C03641=1096.740,305.564,-82.247,178.244,19.160,152.472
C03642=1096.746,305.813,-82.279,178.248,19.162,152.472
C03643=1096.752,306.060,-82.310,178.251,19.165,152.472
C03644=1096.757,306.309,-82.341,178.254,19.167,152.472
C03645=1096.763,306.556,-82.371,178.257,19.170,152.472
C03646=1096.769,306.805,-82.402,178.261,19.172,152.472
C03647=1096.775,307.052,-82.434,178.264,19.175,152.472
C03648=1096.780,307.301,-82.464,178.267,19.177,152.472
C03649=1096.786,307.548,-82.495,178.270,19.180,152.472
C03650=1096.792,307.797,-82.527,178.274,19.183,152.472
C03651=1096.797,308.044,-82.557,178.277,19.185,152.472
C03652=1096.802,308.293,-82.588,178.280,19.188,152.472
C03653=1096.808,308.540,-82.620,178.283,19.190,152.472
C03654=1096.814,308.789,-82.651,178.286,19.193,152.472
C03655=1096.819,309.037,-82.681,178.290,19.195,152.472
C03656=1096.825,309.284,-82.713,178.293,19.197,152.472
C03657=1096.831,309.533,-82.744,178.296,19.200,152.472
C03658=1096.837,309.780,-82.775,178.300,19.203,152.472
C03659=1096.842,310.028,-82.806,178.303,19.206,152.472
C03660=1096.848,310.276,-82.838,178.306,19.208,152.472
C03661=1096.854,310.524,-82.868,178.309,19.211,152.472
C03662=1096.860,310.772,-82.900,178.312,19.213,152.472
C03663=1096.866,311.020,-82.931,178.315,19.215,152.472
C03664=1096.871,311.268,-82.962,178.318,19.218,152.472
C03665=1096.877,311.517,-82.994,178.322,19.221,152.473
C03666=1096.883,311.764,-83.025,178.325,19.223,152.472
C03667=1096.888,312.012,-83.056,178.328,19.226,152.473
C03668=1096.894,312.260,-83.088,178.332,19.229,152.473
C03669=1096.900,312.507,-83.119,178.335,19.231,152.473
C03670=1096.906,312.756,-83.150,178.338,19.234,152.473
C03671=1096.912,313.003,-83.181,178.341,19.237,152.473
C03672=1096.918,313.252,-83.213,178.344,19.239,152.473
C03673=1096.923,313.500,-83.244,178.347,19.241,152.473
C03674=1096.929,313.747,-83.276,178.351,19.244,152.473
C03675=1096.935,313.995,-83.307,178.354,19.247,152.473
C03676=1096.940,314.243,-83.338,178.357,19.249,152.473
C03677=1096.946,314.491,-83.370,178.361,19.252,152.473
C03678=1096.953,314.739,-83.401,178.364,19.255,152.473
C03679=1096.959,314.987,-83.433,178.367,19.258,152.473
C03680=1096.964,315.235,-83.464,178.370,19.260,152.473
C03681=1096.970,315.483,-83.496,178.373,19.263,152.473
C03682=1096.975,315.731,-83.528,178.376,19.265,152.473
C03683=1096.983,316.120,-83.577,178.382,19.270,152.473
C03684=1096.993,316.508,-83.626,178.386,19.274,152.473
C03685=1097.002,316.897,-83.677,178.391,19.279,152.474
C03686=1097.010,317.286,-83.726,178.396,19.283,152.474
C03687=1097.016,317.534,-83.758,178.399,19.286,152.474
C03688=1097.022,317.782,-83.790,178.403,19.289,152.474
C03689=1097.027,318.029,-83.822,178.406,19.291,152.474
C03690=1097.033,318.277,-83.854,178.409,19.295,152.474
C03691=1097.038,318.525,-83.886,178.412,19.297,152.474
C03692=1097.044,318.774,-83.918,178.415,19.300,152.474
C03693=1097.049,319.021,-83.950,178.418,19.303,152.474
C03694=1097.055,319.269,-83.982,178.422,19.306,152.474
C03695=1097.061,319.517,-84.013,178.425,19.308,152.475
C03696=1097.067,319.765,-84.045,178.428,19.311,152.475
C03697=1097.072,320.012,-84.077,178.431,19.314,152.475
C03698=1097.078,320.261,-84.109,178.434,19.317,152.475
C03699=1097.083,320.508,-84.141,178.438,19.320,152.475
C03700=1097.089,320.756,-84.173,178.441,19.323,152.475
C03701=1097.094,321.004,-84.205,178.444,19.326,152.475
C03702=1097.100,321.252,-84.237,178.446,19.329,152.475
C03703=1097.105,321.500,-84.269,178.450,19.331,152.475
C03704=1097.111,321.748,-84.301,178.453,19.335,152.476
C03705=1097.117,321.996,-84.332,178.456,19.337,152.476
C03706=1097.123,322.243,-84.365,178.459,19.340,152.476
C03707=1097.128,322.492,-84.398,178.462,19.343,152.476
C03708=1097.134,322.739,-84.429,178.465,19.346,152.476
C03709=1097.140,322.988,-84.461,178.469,19.349,152.476
C03710=1097.145,323.235,-84.493,178.472,19.352,152.476
C03711=1097.151,323.483,-84.526,178.475,19.355,152.476
C03712=1097.156,323.731,-84.558,178.478,19.357,152.477
C03713=1097.162,323.979,-84.590,178.481,19.360,152.477
C03714=1097.168,324.227,-84.622,178.485,19.364,152.477
C03715=1097.174,324.474,-84.655,178.488,19.366,152.477
C03716=1097.180,324.722,-84.687,178.491,19.369,152.477
C03717=1097.185,324.971,-84.719,178.494,19.372,152.477
C03718=1097.191,325.218,-84.752,178.498,19.375,152.477
C03719=1097.196,325.466,-84.784,178.500,19.379,152.478
C03720=1097.202,325.714,-84.816,178.504,19.381,152.478
C03721=1097.208,325.962,-84.849,178.507,19.384,152.478
C03722=1097.214,326.210,-84.881,178.510,19.388,152.478
C03723=1097.220,326.457,-84.913,178.513,19.390,152.478
C03724=1097.225,326.705,-84.946,178.516,19.393,152.478
C03725=1097.231,326.954,-84.978,178.519,19.396,152.478
C03726=1097.237,327.200,-85.010,178.523,19.399,152.478
C03727=1097.243,327.449,-85.042,178.526,19.402,152.479
C03728=1097.248,327.697,-85.076,178.529,19.405,152.479
C03729=1097.254,327.945,-85.108,178.532,19.408,152.479
C03730=1097.260,328.192,-85.140,178.536,19.411,152.479
C03731=1097.265,328.440,-85.173,178.539,19.414,152.479
C03732=1097.271,328.688,-85.206,178.541,19.417,152.479
C03733=1097.278,328.935,-85.238,178.544,19.420,152.479
C03734=1097.283,329.184,-85.271,178.548,19.423,152.480
C03735=1097.292,329.565,-85.320,178.553,19.428,152.480
C03736=1097.301,329.947,-85.371,178.558,19.433,152.480
C03737=1097.310,330.328,-85.422,178.563,19.438,152.480
C03738=1097.319,330.711,-85.472,178.567,19.442,152.481
C03739=1097.325,330.958,-85.504,178.570,19.445,152.481
C03740=1097.330,331.206,-85.537,178.574,19.448,152.481
C03741=1097.336,331.454,-85.570,178.577,19.451,152.481
C03742=1097.342,331.702,-85.603,178.580,19.454,152.481
C03743=1097.348,331.949,-85.636,178.584,19.458,152.481
C03744=1097.354,332.197,-85.668,178.586,19.461,152.482
C03745=1097.360,332.445,-85.701,178.589,19.464,152.482
C03746=1097.365,332.692,-85.734,178.593,19.467,152.482
C03747=1097.371,332.940,-85.767,178.596,19.470,152.482
C03748=1097.376,333.189,-85.800,178.599,19.473,152.482
C03749=1097.382,333.436,-85.833,178.602,19.477,152.483
C03750=1097.388,333.684,-85.866,178.605,19.480,152.483
C03751=1097.394,333.932,-85.899,178.608,19.483,152.483
C03752=1097.400,334.180,-85.932,178.612,19.487,152.483
C03753=1097.405,334.427,-85.965,178.615,19.489,152.483
C03754=1097.410,334.675,-85.998,178.618,19.493,152.484
C03755=1097.417,334.922,-86.031,178.621,19.496,152.484
C03756=1097.422,335.170,-86.064,178.624,19.499,152.484
C03757=1097.428,335.418,-86.097,178.627,19.502,152.484
C03758=1097.433,335.667,-86.130,178.630,19.506,152.485
C03759=1097.439,335.914,-86.163,178.633,19.509,152.485
C03760=1097.445,336.162,-86.196,178.636,19.512,152.485
C03761=1097.450,336.410,-86.229,178.640,19.516,152.485
C03762=1097.456,336.656,-86.263,178.643,19.519,152.485
C03763=1097.462,336.904,-86.296,178.646,19.523,152.486
C03764=1097.467,337.152,-86.329,178.649,19.526,152.486
C03765=1097.473,337.400,-86.363,178.652,19.529,152.486
C03766=1097.479,337.648,-86.395,178.655,19.533,152.486
C03767=1097.485,337.895,-86.429,178.658,19.536,152.487
C03768=1097.490,338.143,-86.462,178.661,19.539,152.487
C03769=1097.496,338.391,-86.495,178.665,19.542,152.487
C03770=1097.502,338.639,-86.528,178.668,19.546,152.487
C03771=1097.508,338.886,-86.562,178.671,19.550,152.488
C03772=1097.514,339.134,-86.595,178.674,19.553,152.488
C03773=1097.519,339.382,-86.629,178.677,19.556,152.488
C03774=1097.525,339.630,-86.662,178.680,19.560,152.488
C03775=1097.530,339.878,-86.695,178.683,19.563,152.489
C03776=1097.536,340.125,-86.730,178.686,19.567,152.489
C03777=1097.542,340.373,-86.763,178.689,19.570,152.489
C03778=1097.547,340.621,-86.796,178.693,19.573,152.489
C03779=1097.553,340.869,-86.830,178.696,19.577,152.490
C03780=1097.559,341.116,-86.863,178.698,19.580,152.490
C03781=1097.565,341.364,-86.896,178.702,19.584,152.490
C03782=1097.571,341.612,-86.930,178.705,19.587,152.491
C03783=1097.576,341.859,-86.964,178.708,19.591,152.491
C03784=1097.582,342.107,-86.997,178.711,19.594,152.491
C03785=1097.588,342.354,-87.031,178.714,19.598,152.492
C03786=1097.593,342.602,-87.064,178.717,19.601,152.492
C03787=1097.602,342.979,-87.116,178.722,19.607,152.492
C03788=1097.611,343.353,-87.167,178.727,19.612,152.493
C03789=1097.619,343.729,-87.218,178.731,19.617,152.493
C03790=1097.629,344.105,-87.269,178.736,19.623,152.494
C03791=1097.634,344.353,-87.304,178.740,19.626,152.494
C03792=1097.640,344.601,-87.337,178.742,19.630,152.494
C03793=1097.645,344.848,-87.371,178.746,19.634,152.494
C03794=1097.651,345.096,-87.404,178.748,19.637,152.495
C03795=1097.657,345.343,-87.438,178.751,19.641,152.495
C03796=1097.662,345.591,-87.472,178.755,19.644,152.495
C03797=1097.668,345.838,-87.506,178.757,19.648,152.496
C03798=1097.674,346.085,-87.540,178.761,19.652,152.496
C03799=1097.680,346.334,-87.573,178.764,19.655,152.496
C03800=1097.685,346.582,-87.608,178.767,19.659,152.497
C03801=1097.691,346.829,-87.642,178.770,19.663,152.497
C03802=1097.697,347.077,-87.675,178.773,19.666,152.497
C03803=1097.703,347.324,-87.710,178.776,19.670,152.498
C03804=1097.708,347.571,-87.744,178.779,19.674,152.498
C03805=1097.714,347.819,-87.778,178.782,19.677,152.499
C03806=1097.720,348.068,-87.812,178.785,19.681,152.499
C03807=1097.726,348.315,-87.846,178.789,19.685,152.499
C03808=1097.731,348.562,-87.880,178.791,19.689,152.500
C03809=1097.737,348.809,-87.914,178.795,19.693,152.500
C03810=1097.742,349.058,-87.948,178.798,19.696,152.500
C03811=1097.748,349.305,-87.982,178.801,19.700,152.501
C03812=1097.754,349.553,-88.017,178.804,19.704,152.501
C03813=1097.760,349.801,-88.051,178.807,19.708,152.501
C03814=1097.765,350.048,-88.085,178.810,19.712,152.502
C03815=1097.771,350.295,-88.119,178.813,19.716,152.502
C03816=1097.776,350.543,-88.154,178.816,19.719,152.503
C03817=1097.783,350.791,-88.188,178.819,19.723,152.503
C03818=1097.789,351.038,-88.222,178.822,19.727,152.503
C03819=1097.794,351.286,-88.257,178.825,19.731,152.504
C03820=1097.800,351.533,-88.291,178.828,19.735,152.504
C03821=1097.806,351.781,-88.326,178.831,19.738,152.504
C03822=1097.811,352.028,-88.360,178.834,19.742,152.505
C03823=1097.817,352.276,-88.394,178.837,19.746,152.505
C03824=1097.823,352.523,-88.428,178.840,19.750,152.506
C03825=1097.829,352.771,-88.463,178.843,19.754,152.506
C03826=1097.835,353.019,-88.497,178.846,19.758,152.506
C03827=1097.841,353.266,-88.531,178.850,19.762,152.507
C03828=1097.846,353.513,-88.566,178.852,19.766,152.507
C03829=1097.852,353.761,-88.600,178.856,19.770,152.508
C03830=1097.857,354.009,-88.635,178.858,19.773,152.508
C03831=1097.863,354.256,-88.669,178.862,19.777,152.508
C03832=1097.869,354.504,-88.705,178.865,19.782,152.509
C03833=1097.875,354.751,-88.739,178.867,19.785,152.509
C03834=1097.880,354.999,-88.774,178.871,19.789,152.510
C03835=1097.886,355.246,-88.808,178.873,19.793,152.510
C03836=1097.892,355.494,-88.843,178.877,19.798,152.511
C03837=1097.897,355.741,-88.878,178.880,19.802,152.511
C03838=1097.903,355.989,-88.912,178.883,19.806,152.512
C03839=1097.911,356.367,-88.965,178.887,19.812,152.512
C03840=1097.921,356.745,-89.018,178.891,19.818,152.513
C03841=1097.930,357.123,-89.071,178.897,19.825,152.514
C03842=1097.938,357.501,-89.125,178.902,19.831,152.514
C03843=1097.944,357.749,-89.160,178.904,19.835,152.515
C03844=1097.950,357.996,-89.194,178.907,19.839,152.515
C03845=1097.955,358.244,-89.229,178.911,19.843,152.516
C03846=1097.962,358.491,-89.264,178.913,19.847,152.516
C03847=1097.967,358.738,-89.299,178.916,19.851,152.517
C03848=1097.973,358.986,-89.334,178.920,19.856,152.517
C03849=1097.979,359.233,-89.369,178.922,19.860,152.518
C03850=1097.985,359.481,-89.404,178.925,19.864,152.518
C03851=1097.990,359.728,-89.439,178.929,19.868,152.519
C03852=1097.997,359.976,-89.474,178.931,19.872,152.519
C03853=1098.002,360.223,-89.509,178.934,19.877,152.520
C03854=1098.007,360.470,-89.544,178.938,19.881,152.520
C03855=1098.013,360.719,-89.579,178.940,19.885,152.521
C03856=1098.019,360.965,-89.614,178.943,19.889,152.521
C03857=1098.025,361.213,-89.650,178.946,19.894,152.522
C03858=1098.030,361.461,-89.684,178.949,19.898,152.522
C03859=1098.036,361.708,-89.720,178.952,19.902,152.523
C03860=1098.042,361.955,-89.755,178.955,19.907,152.523
C03861=1098.048,362.203,-89.789,178.958,19.911,152.524
C03862=1098.054,362.450,-89.825,178.961,19.915,152.524
C03863=1098.059,362.697,-89.860,178.964,19.920,152.525
C03864=1098.065,362.945,-89.895,178.967,19.924,152.525
C03865=1098.070,363.192,-89.931,178.969,19.928,152.526
C03866=1098.077,363.440,-89.966,178.973,19.932,152.526
C03867=1098.082,363.687,-90.001,178.976,19.937,152.527
C03868=1098.088,363.934,-90.037,178.979,19.941,152.527
C03869=1098.093,364.182,-90.072,178.982,19.945,152.528
C03870=1098.100,364.430,-90.107,178.984,19.950,152.529
C03871=1098.105,364.677,-90.143,178.988,19.955,152.529
C03872=1098.111,364.924,-90.179,178.991,19.959,152.530
C03873=1098.117,365.171,-90.213,178.993,19.963,152.530
C03874=1098.123,365.419,-90.249,178.996,19.968,152.531
C03875=1098.129,365.666,-90.284,178.999,19.973,152.531
C03876=1098.135,365.913,-90.320,179.003,19.977,152.532
C03877=1098.141,366.161,-90.356,179.005,19.981,152.532
C03878=1098.146,366.409,-90.391,179.008,19.986,152.533
C03879=1098.152,366.656,-90.426,179.011,19.990,152.534
C03880=1098.158,366.903,-90.462,179.014,19.995,152.534
C03881=1098.163,367.151,-90.499,179.017,19.999,152.535
C03882=1098.168,367.398,-90.534,179.020,20.004,152.535
C03883=1098.174,367.645,-90.570,179.023,20.009,152.536
C03884=1098.180,367.892,-90.605,179.026,20.014,152.537
C03885=1098.186,368.140,-90.641,179.029,20.019,152.537
C03886=1098.191,368.387,-90.676,179.031,20.022,152.538
C03887=1098.197,368.635,-90.712,179.034,20.027,152.539
C03888=1098.203,368.882,-90.747,179.037,20.032,152.539
C03889=1098.209,369.129,-90.783,179.040,20.037,152.540
C03890=1098.215,369.377,-90.819,179.043,20.042,152.540
C03891=1098.223,369.770,-90.876,179.047,20.049,152.541
C03892=1098.232,370.163,-90.933,179.052,20.056,152.542
C03893=1098.242,370.556,-90.990,179.057,20.064,152.543
C03894=1098.251,370.949,-91.047,179.061,20.072,152.545
C03895=1098.256,371.197,-91.083,179.064,20.076,152.545
C03896=1098.263,371.444,-91.119,179.067,20.081,152.546
C03897=1098.268,371.691,-91.155,179.070,20.086,152.546
C03898=1098.274,371.938,-91.191,179.073,20.091,152.547
C03899=1098.280,372.185,-91.227,179.076,20.096,152.548
C03900=1098.285,372.433,-91.263,179.078,20.100,152.548
C03901=1098.291,372.680,-91.299,179.081,20.105,152.549
C03902=1098.297,372.927,-91.335,179.084,20.110,152.550
C03903=1098.304,373.174,-91.372,179.087,20.115,152.550
C03904=1098.309,373.421,-91.407,179.090,20.120,152.551
C03905=1098.315,373.669,-91.443,179.093,20.125,152.552
C03906=1098.321,373.916,-91.480,179.096,20.130,152.553
C03907=1098.326,374.163,-91.515,179.099,20.135,152.553
C03908=1098.333,374.410,-91.552,179.101,20.139,152.554
C03909=1098.338,374.658,-91.589,179.104,20.144,152.555
C03910=1098.344,374.906,-91.624,179.107,20.149,152.555
C03911=1098.349,375.152,-91.661,179.110,20.154,152.556
C03912=1098.355,375.400,-91.697,179.113,20.159,152.557
C03913=1098.362,375.647,-91.733,179.116,20.164,152.558
C03914=1098.366,375.894,-91.769,179.119,20.169,152.558
C03915=1098.373,376.141,-91.806,179.122,20.175,152.559
C03916=1098.378,376.389,-91.843,179.125,20.180,152.560
C03917=1098.384,376.636,-91.878,179.127,20.185,152.561
C03918=1098.389,376.883,-91.915,179.130,20.190,152.561
C03919=1098.396,377.130,-91.951,179.133,20.195,152.562
C03920=1098.401,377.377,-91.988,179.135,20.200,152.563
C03921=1098.407,377.625,-92.024,179.138,20.205,152.564
C03922=1098.412,377.872,-92.061,179.141,20.210,152.564
C03923=1098.419,378.119,-92.097,179.144,20.215,152.565
C03924=1098.424,378.366,-92.134,179.147,20.221,152.566
C03925=1098.431,378.613,-92.171,179.150,20.226,152.567
C03926=1098.435,378.860,-92.207,179.152,20.231,152.568
C03927=1098.442,379.108,-92.243,179.155,20.236,152.568
C03928=1098.447,379.355,-92.280,179.158,20.242,152.569
C03929=1098.453,379.602,-92.317,179.161,20.247,152.570
C03930=1098.459,379.849,-92.354,179.164,20.252,152.571
C03931=1098.465,380.096,-92.390,179.167,20.257,152.571
C03932=1098.470,380.343,-92.427,179.169,20.262,152.572
C03933=1098.477,380.590,-92.463,179.172,20.268,152.573
C03934=1098.482,380.837,-92.500,179.175,20.273,152.574
C03935=1098.488,381.085,-92.537,179.178,20.278,152.575
C03936=1098.494,381.332,-92.574,179.181,20.284,152.576
C03937=1098.500,381.579,-92.611,179.183,20.289,152.576
C03938=1098.506,381.826,-92.647,179.186,20.294,152.577
C03939=1098.512,382.074,-92.684,179.189,20.300,152.578
C03940=1098.517,382.320,-92.721,179.191,20.305,152.579
C03941=1098.523,382.567,-92.757,179.194,20.311,152.580
C03942=1098.529,382.815,-92.794,179.197,20.316,152.581
C03943=1098.534,383.025,-92.826,179.200,20.321,152.581
C03944=1098.539,383.235,-92.858,179.202,20.326,152.582
C03945=1098.544,383.445,-92.889,179.204,20.330,152.583
C03946=1098.548,383.655,-92.921,179.206,20.335,152.584
C03947=1098.553,383.865,-92.952,179.209,20.340,152.584
C03948=1098.559,384.075,-92.983,179.211,20.344,152.585
C03949=1098.563,384.286,-93.014,179.213,20.349,152.586
C03950=1098.568,384.495,-93.046,179.216,20.354,152.587
C03951=1098.574,384.742,-93.083,179.219,20.360,152.588
C03952=1098.580,384.990,-93.120,179.221,20.365,152.589
C03953=1098.585,385.237,-93.157,179.224,20.371,152.589
C03954=1098.591,385.484,-93.195,179.227,20.376,152.590
C03955=1098.597,385.731,-93.232,179.229,20.382,152.591
C03956=1098.603,385.978,-93.269,179.232,20.387,152.592
C03957=1098.609,386.225,-93.306,179.235,20.393,152.593
C03958=1098.615,386.472,-93.343,179.238,20.399,152.594
C03959=1098.620,386.720,-93.380,179.241,20.405,152.595
C03960=1098.626,386.966,-93.418,179.243,20.411,152.596
C03961=1098.632,387.214,-93.455,179.246,20.417,152.597
C03962=1098.638,387.461,-93.493,179.249,20.422,152.598
C03963=1098.643,387.708,-93.530,179.251,20.428,152.599
C03964=1098.649,387.955,-93.568,179.254,20.433,152.600
C03965=1098.655,388.202,-93.604,179.257,20.440,152.601
C03966=1098.661,388.448,-93.642,179.260,20.445,152.601
C03967=1098.667,388.696,-93.679,179.262,20.451,152.603
C03968=1098.673,388.943,-93.717,179.265,20.457,152.604
C03969=1098.678,389.190,-93.754,179.268,20.463,152.605
C03970=1098.684,389.437,-93.792,179.270,20.469,152.605
C03971=1098.690,389.683,-93.829,179.274,20.475,152.606
C03972=1098.696,389.931,-93.866,179.276,20.481,152.607
C03973=1098.702,390.177,-93.904,179.279,20.487,152.608
C03974=1098.708,390.424,-93.942,179.281,20.492,152.609
C03975=1098.713,390.672,-93.979,179.284,20.498,152.610
C03976=1098.719,390.918,-94.017,179.286,20.504,152.612
C03977=1098.726,391.166,-94.055,179.290,20.511,152.612
C03978=1098.731,391.413,-94.092,179.292,20.516,152.613
C03979=1098.737,391.660,-94.130,179.295,20.522,152.615
C03980=1098.743,391.907,-94.167,179.297,20.528,152.615
C03981=1098.749,392.153,-94.205,179.300,20.534,152.617
C03982=1098.755,392.401,-94.242,179.303,20.541,152.618
C03983=1098.761,392.648,-94.280,179.305,20.547,152.619
C03984=1098.766,392.895,-94.319,179.308,20.553,152.620
C03985=1098.772,393.142,-94.356,179.310,20.559,152.621
C03986=1098.778,393.389,-94.394,179.313,20.566,152.622
C03987=1098.784,393.635,-94.432,179.316,20.572,152.623
C03988=1098.790,393.882,-94.470,179.318,20.578,152.624
C03989=1098.795,394.131,-94.508,179.321,20.584,152.625
C03990=1098.801,394.377,-94.545,179.324,20.590,152.626
C03991=1098.807,394.624,-94.583,179.326,20.596,152.627
C03992=1098.813,394.871,-94.621,179.329,20.603,152.629
C03993=1098.818,395.118,-94.659,179.331,20.609,152.630
C03994=1098.825,395.365,-94.697,179.334,20.616,152.631
C03995=1098.831,395.612,-94.735,179.337,20.622,152.632
C03996=1098.836,395.859,-94.773,179.339,20.628,152.633
C03997=1098.842,396.106,-94.811,179.342,20.635,152.634
C03998=1098.848,396.353,-94.849,179.344,20.641,152.635
C03999=1098.853,396.569,-94.883,179.347,20.647,152.636
C04000=1098.858,396.785,-94.917,179.349,20.652,152.637
C04001=1098.863,397.002,-94.949,179.351,20.658,152.638
C04002=1098.868,397.219,-94.983,179.354,20.664,152.639
C04003=1098.874,397.434,-95.017,179.356,20.669,152.640
C04004=1098.879,397.651,-95.051,179.358,20.675,152.641
C04005=1098.884,397.868,-95.083,179.361,20.681,152.642
C04006=1098.888,398.084,-95.117,179.362,20.686,152.643
C04007=1098.895,398.331,-95.155,179.365,20.693,152.645
C04008=1098.900,398.578,-95.194,179.368,20.700,152.646
C04009=1098.906,398.825,-95.232,179.370,20.706,152.647
C04010=1098.913,399.072,-95.270,179.373,20.713,152.648
C04011=1098.918,399.319,-95.309,179.375,20.720,152.649
C04012=1098.924,399.565,-95.347,179.377,20.726,152.651
C04013=1098.930,399.813,-95.386,179.380,20.733,152.652
C04014=1098.936,400.060,-95.424,179.383,20.740,152.653
C04015=1098.941,400.307,-95.462,179.386,20.747,152.654
C04016=1098.947,400.554,-95.501,179.388,20.753,152.656
C04017=1098.953,400.801,-95.539,179.390,20.760,152.657
C04018=1098.959,401.048,-95.578,179.393,20.767,152.658
C04019=1098.965,401.294,-95.616,179.395,20.774,152.659
C04020=1098.970,401.542,-95.655,179.398,20.781,152.661
C04021=1098.976,401.789,-95.694,179.400,20.788,152.662
C04022=1098.982,402.035,-95.732,179.404,20.795,152.663
C04023=1098.988,402.283,-95.771,179.406,20.802,152.665
C04024=1098.994,402.529,-95.809,179.408,20.808,152.666
C04025=1098.999,402.776,-95.848,179.411,20.815,152.667
C04026=1099.005,403.023,-95.887,179.413,20.822,152.668
C04027=1099.011,403.270,-95.925,179.416,20.829,152.670
C04028=1099.018,403.517,-95.965,179.418,20.836,152.671
C04029=1099.023,403.764,-96.003,179.421,20.844,152.672
C04030=1099.030,404.011,-96.042,179.423,20.850,152.674
C04031=1099.035,404.258,-96.080,179.426,20.858,152.675
C04032=1099.041,404.505,-96.120,179.428,20.865,152.676
C04033=1099.047,404.751,-96.158,179.431,20.872,152.678
C04034=1099.053,404.999,-96.197,179.434,20.879,152.679
C04035=1099.058,405.245,-96.236,179.436,20.886,152.680
C04036=1099.064,405.492,-96.275,179.439,20.893,152.682
C04037=1099.070,405.738,-96.314,179.441,20.900,152.683
C04038=1099.076,405.986,-96.352,179.444,20.908,152.685
C04039=1099.082,406.233,-96.392,179.445,20.915,152.686
C04040=1099.088,406.480,-96.431,179.448,20.923,152.687
C04041=1099.093,406.726,-96.470,179.450,20.930,152.689
C04042=1099.099,406.973,-96.509,179.453,20.937,152.690
C04043=1099.105,407.220,-96.549,179.456,20.945,152.692
C04044=1099.111,407.467,-96.587,179.458,20.952,152.693
C04045=1099.117,407.714,-96.626,179.461,20.959,152.694
C04046=1099.123,407.961,-96.665,179.463,20.967,152.696
C04047=1099.129,408.208,-96.705,179.465,20.974,152.697
C04048=1099.134,408.454,-96.744,179.468,20.982,152.699
C04049=1099.140,408.701,-96.783,179.471,20.990,152.700
C04050=1099.146,408.948,-96.822,179.473,20.997,152.702
C04051=1099.152,409.195,-96.862,179.475,21.005,152.703
C04052=1099.158,409.441,-96.901,179.478,21.013,152.705
C04053=1099.164,409.689,-96.940,179.480,21.020,152.706
C04054=1099.170,409.936,-96.980,179.483,21.028,152.708
C04055=1099.175,410.151,-97.014,179.485,21.035,152.709
C04056=1099.179,410.368,-97.049,179.487,21.041,152.710
C04057=1099.184,410.585,-97.084,179.489,21.048,152.712
C04058=1099.190,410.801,-97.118,179.491,21.055,152.713
C04059=1099.195,411.018,-97.152,179.493,21.062,152.715
C04060=1099.200,411.235,-97.187,179.495,21.069,152.716
C04061=1099.205,411.451,-97.221,179.498,21.075,152.717
C04062=1099.211,411.668,-97.256,179.500,21.082,152.719
C04063=1099.216,411.914,-97.296,179.502,21.090,152.720
C04064=1099.222,412.162,-97.335,179.505,21.098,152.722
C04065=1099.228,412.408,-97.376,179.507,21.106,152.723
C04066=1099.234,412.654,-97.415,179.509,21.114,152.725
C04067=1099.240,412.902,-97.454,179.512,21.122,152.726
C04068=1099.246,413.148,-97.494,179.514,21.130,152.728
C04069=1099.252,413.395,-97.533,179.517,21.138,152.730
C04070=1099.258,413.642,-97.573,179.520,21.146,152.731
C04071=1099.263,413.889,-97.614,179.521,21.154,152.733
C04072=1099.269,414.136,-97.653,179.524,21.162,152.734
C04073=1099.275,414.381,-97.693,179.526,21.170,152.736
C04074=1099.281,414.629,-97.732,179.529,21.179,152.738
C04075=1099.288,414.875,-97.772,179.531,21.187,152.739
C04076=1099.294,415.122,-97.812,179.534,21.195,152.741
C04077=1099.299,415.369,-97.852,179.536,21.203,152.743
C04078=1099.305,415.616,-97.892,179.538,21.211,152.744
C04079=1099.311,415.862,-97.932,179.541,21.219,152.746
C04080=1099.317,416.109,-97.971,179.543,21.228,152.748
C04081=1099.324,416.356,-98.011,179.546,21.236,152.749
C04082=1099.329,416.603,-98.051,179.548,21.245,152.751
C04083=1099.335,416.849,-98.091,179.551,21.253,152.753
C04084=1099.340,417.096,-98.132,179.553,21.262,152.754
C04085=1099.346,417.343,-98.171,179.555,21.270,152.756
C04086=1099.353,417.589,-98.211,179.558,21.279,152.758
C04087=1099.358,417.836,-98.252,179.560,21.287,152.760
C04088=1099.364,418.082,-98.292,179.562,21.296,152.761
C04089=1099.370,418.330,-98.332,179.565,21.305,152.763
C04090=1099.376,418.576,-98.372,179.567,21.313,152.765
C04091=1099.382,418.823,-98.412,179.569,21.322,152.767
C04092=1099.388,419.069,-98.453,179.572,21.331,152.769
C04093=1099.394,419.316,-98.493,179.574,21.339,152.770
C04094=1099.399,419.563,-98.533,179.577,21.348,152.772
C04095=1099.405,419.809,-98.573,179.579,21.357,152.774
C04096=1099.411,420.056,-98.614,179.581,21.365,152.776
C04097=1099.417,420.302,-98.654,179.583,21.374,152.778
C04098=1099.423,420.549,-98.695,179.586,21.383,152.779
C04099=1099.430,420.796,-98.735,179.588,21.392,152.781
C04100=1099.435,421.043,-98.775,179.590,21.401,152.783
C04101=1099.442,421.289,-98.816,179.593,21.410,152.785
C04102=1099.447,421.536,-98.856,179.595,21.419,152.787
C04103=1099.454,421.783,-98.897,179.597,21.428,152.789
C04104=1099.459,422.029,-98.937,179.599,21.436,152.791
C04105=1099.466,422.276,-98.977,179.602,21.446,152.792
C04106=1099.471,422.522,-99.018,179.605,21.455,152.794
C04107=1099.477,422.768,-99.059,179.607,21.464,152.796
C04108=1099.483,423.015,-99.099,179.609,21.473,152.798
C04109=1099.489,423.262,-99.140,179.611,21.482,152.800
C04110=1099.494,423.508,-99.181,179.613,21.491,152.802
C04111=1099.500,423.732,-99.218,179.616,21.500,152.804
C04112=1099.505,423.955,-99.255,179.617,21.508,152.806
C04113=1099.511,424.179,-99.292,179.620,21.517,152.807
C04114=1099.516,424.402,-99.329,179.622,21.525,152.809
C04115=1099.522,424.626,-99.365,179.623,21.534,152.811
C04116=1099.527,424.849,-99.402,179.626,21.543,152.813
C04117=1099.532,425.073,-99.440,179.628,21.551,152.815
C04118=1099.538,425.296,-99.476,179.630,21.559,152.816
C04119=1099.544,425.542,-99.518,179.632,21.569,152.818
C04120=1099.549,425.789,-99.559,179.635,21.579,152.821
C04121=1099.555,426.036,-99.599,179.637,21.588,152.823
C04122=1099.562,426.282,-99.640,179.639,21.598,152.825
C04123=1099.567,426.529,-99.681,179.641,21.607,152.827
C04124=1099.573,426.775,-99.722,179.644,21.617,152.829
C04125=1099.579,427.022,-99.763,179.646,21.627,152.831
C04126=1099.585,427.268,-99.805,179.648,21.636,152.833
C04127=1099.591,427.514,-99.845,179.650,21.647,152.835
C04128=1099.597,427.761,-99.886,179.652,21.656,152.837
C04129=1099.603,428.007,-99.928,179.654,21.666,152.839
C04130=1099.609,428.254,-99.968,179.657,21.676,152.841
C04131=1099.615,428.500,-100.010,179.659,21.686,152.844
C04132=1099.621,428.747,-100.052,179.661,21.695,152.846
C04133=1099.627,428.994,-100.092,179.664,21.706,152.848
C04134=1099.633,429.240,-100.134,179.665,21.716,152.850
C04135=1099.639,429.486,-100.175,179.667,21.726,152.852
C04136=1099.645,429.732,-100.217,179.670,21.736,152.854
C04137=1099.651,429.979,-100.258,179.672,21.746,152.857
C04138=1099.656,430.225,-100.299,179.674,21.756,152.859
C04139=1099.662,430.471,-100.340,179.676,21.766,152.861
C04140=1099.668,430.718,-100.382,179.678,21.776,152.863
C04141=1099.675,430.965,-100.424,179.681,21.787,152.865
C04142=1099.681,431.211,-100.465,179.683,21.797,152.868
C04143=1099.687,431.458,-100.506,179.684,21.807,152.870
C04144=1099.692,431.704,-100.547,179.687,21.818,152.872
C04145=1099.698,431.950,-100.589,179.689,21.828,152.875
C04146=1099.705,432.197,-100.631,179.691,21.838,152.877
C04147=1099.711,432.443,-100.672,179.693,21.849,152.879
C04148=1099.717,432.689,-100.714,179.696,21.859,152.881
C04149=1099.723,432.936,-100.755,179.697,21.870,152.884
C04150=1099.728,433.181,-100.798,179.700,21.881,152.886
C04151=1099.735,433.428,-100.840,179.702,21.891,152.888
C04152=1099.741,433.675,-100.881,179.704,21.902,152.891
C04153=1099.747,433.921,-100.923,179.706,21.913,152.893
C04154=1099.753,434.167,-100.964,179.708,21.924,152.896
C04155=1099.758,434.413,-101.006,179.710,21.934,152.898
C04156=1099.764,434.660,-101.048,179.712,21.945,152.900
C04157=1099.771,434.906,-101.090,179.714,21.956,152.903
C04158=1099.776,435.152,-101.132,179.716,21.967,152.905
C04159=1099.782,435.399,-101.174,179.719,21.978,152.908
C04160=1099.789,435.645,-101.216,179.720,21.989,152.910
C04161=1099.794,435.891,-101.258,179.722,22.000,152.913
C04162=1099.800,436.138,-101.300,179.724,22.011,152.915
C04163=1099.806,436.383,-101.342,179.726,22.022,152.918
C04164=1099.812,436.630,-101.384,179.729,22.034,152.920
C04165=1099.818,436.877,-101.426,179.730,22.045,152.923
C04166=1099.824,437.122,-101.468,179.733,22.056,152.925
C04167=1099.832,437.464,-101.527,179.735,22.071,152.929
C04168=1099.841,437.805,-101.585,179.738,22.087,152.932
C04169=1099.849,438.146,-101.643,179.741,22.103,152.936
C04170=1099.858,438.488,-101.702,179.744,22.119,152.939
C04171=1099.864,438.734,-101.744,179.745,22.130,152.942
C04172=1099.870,438.981,-101.787,179.747,22.142,152.945
C04173=1099.876,439.226,-101.829,179.750,22.154,152.947
C04174=1099.882,439.474,-101.871,179.752,22.165,152.950
C04175=1099.888,439.719,-101.914,179.753,22.177,152.953
C04176=1099.894,439.965,-101.956,179.755,22.188,152.955
C04177=1099.900,440.211,-101.999,179.757,22.200,152.958
C04178=1099.906,440.457,-102.040,179.760,22.212,152.961
C04179=1099.912,440.704,-102.084,179.761,22.224,152.963
C04180=1099.918,440.950,-102.126,179.763,22.236,152.966
C04181=1099.925,441.196,-102.169,179.765,22.248,152.969
C04182=1099.930,441.442,-102.212,179.767,22.260,152.971
C04183=1099.937,441.688,-102.254,179.768,22.272,152.974
C04184=1099.943,441.934,-102.297,179.771,22.284,152.977
C04185=1099.948,442.181,-102.339,179.772,22.296,152.980
C04186=1099.955,442.427,-102.381,179.775,22.308,152.983
C04187=1099.960,442.673,-102.424,179.777,22.321,152.985
C04188=1099.966,442.920,-102.467,179.779,22.333,152.988
C04189=1099.973,443.165,-102.510,179.780,22.345,152.991
C04190=1099.979,443.412,-102.553,179.782,22.357,152.994
C04191=1099.985,443.657,-102.596,179.783,22.370,152.997
C04192=1099.991,443.904,-102.639,179.786,22.382,153.000
C04193=1099.997,444.149,-102.681,179.786,22.395,153.003
C04194=1100.003,444.396,-102.725,179.788,22.407,153.006
C04195=1100.009,444.642,-102.767,179.789,22.419,153.009
C04196=1100.015,444.888,-102.811,179.790,22.432,153.012
C04197=1100.022,445.135,-102.853,179.791,22.444,153.014
C04198=1100.027,445.380,-102.897,179.792,22.456,153.017
C04199=1100.033,445.626,-102.940,179.792,22.469,153.021
C04200=1100.039,445.872,-102.982,179.793,22.481,153.024
C04201=1100.045,446.119,-103.026,179.793,22.493,153.027
C04202=1100.052,446.365,-103.069,179.794,22.506,153.030
C04203=1100.057,446.611,-103.112,179.794,22.518,153.033
C04204=1100.063,446.857,-103.155,179.794,22.530,153.036
C04205=1100.069,447.103,-103.199,179.794,22.543,153.039
C04206=1100.075,447.349,-103.242,179.793,22.554,153.042
C04207=1100.081,447.596,-103.285,179.793,22.567,153.045
C04208=1100.088,447.841,-103.328,179.792,22.579,153.049
C04209=1100.094,448.087,-103.371,179.792,22.591,153.052
C04210=1100.100,448.333,-103.415,179.791,22.603,153.055
C04211=1100.106,448.579,-103.458,179.790,22.615,153.058
C04212=1100.112,448.826,-103.501,179.789,22.627,153.061
C04213=1100.118,449.072,-103.545,179.788,22.639,153.065
C04214=1100.124,449.318,-103.587,179.787,22.652,153.068
C04215=1100.130,449.564,-103.631,179.786,22.664,153.071
C04216=1100.136,449.810,-103.674,179.784,22.676,153.074
C04217=1100.142,450.056,-103.718,179.783,22.688,153.078
C04218=1100.148,450.302,-103.761,179.781,22.699,153.081
C04219=1099.752,450.294,-103.910,179.716,22.920,153.146
C04220=1099.745,450.048,-103.866,179.718,22.909,153.143
C04221=1099.739,449.802,-103.822,179.719,22.896,153.140
C04222=1099.733,449.555,-103.779,179.720,22.884,153.137
C04223=1099.726,449.310,-103.736,179.722,22.872,153.133
C04224=1099.720,449.064,-103.693,179.723,22.860,153.130
C04225=1099.715,448.817,-103.649,179.724,22.847,153.127
C04226=1099.708,448.571,-103.606,179.725,22.835,153.124
C04227=1099.703,448.325,-103.562,179.726,22.823,153.120
C04228=1099.697,448.079,-103.519,179.727,22.811,153.117
C04229=1099.690,447.833,-103.475,179.727,22.798,153.114
C04230=1099.685,447.587,-103.432,179.728,22.786,153.111
C04231=1099.677,447.341,-103.389,179.727,22.774,153.108
C04232=1099.671,447.095,-103.346,179.728,22.761,153.104
C04233=1099.665,446.849,-103.303,179.728,22.750,153.101
C04234=1099.659,446.603,-103.259,179.728,22.737,153.098
C04235=1099.653,446.356,-103.216,179.728,22.725,153.095
C04236=1099.647,446.111,-103.173,179.727,22.712,153.092
C04237=1099.641,445.864,-103.130,179.727,22.700,153.089
C04238=1099.635,445.618,-103.087,179.726,22.687,153.086
C04239=1099.629,445.372,-103.043,179.726,22.675,153.083
C04240=1099.623,445.126,-103.000,179.725,22.663,153.080
C04241=1099.617,444.879,-102.957,179.724,22.651,153.077
C04242=1099.611,444.634,-102.915,179.723,22.638,153.074
C04243=1099.604,444.388,-102.871,179.722,22.626,153.071
C04244=1099.599,444.142,-102.828,179.720,22.613,153.068
C04245=1099.593,443.895,-102.785,179.719,22.601,153.065
C04246=1099.587,443.649,-102.742,179.717,22.588,153.062
C04247=1099.580,443.403,-102.700,179.715,22.576,153.059
C04248=1099.575,443.158,-102.656,179.713,22.563,153.056
C04249=1099.569,442.911,-102.613,179.711,22.550,153.053
C04250=1099.563,442.665,-102.570,179.710,22.539,153.051
C04251=1099.556,442.419,-102.528,179.708,22.526,153.048
C04252=1099.550,442.172,-102.484,179.705,22.514,153.045
C04253=1099.544,441.927,-102.442,179.703,22.501,153.042
C04254=1099.538,441.680,-102.399,179.701,22.489,153.039
C04255=1099.532,441.434,-102.356,179.699,22.477,153.037
C04256=1099.526,441.189,-102.314,179.698,22.466,153.034
C04257=1099.520,440.942,-102.271,179.696,22.453,153.031
C04258=1099.515,440.696,-102.229,179.693,22.441,153.028
C04259=1099.508,440.449,-102.186,179.691,22.429,153.026
C04260=1099.502,440.203,-102.144,179.690,22.418,153.023
C04261=1099.495,439.957,-102.101,179.688,22.406,153.020
C04262=1099.490,439.711,-102.058,179.685,22.394,153.018
C04263=1099.483,439.465,-102.016,179.683,22.382,153.015
C04264=1099.478,439.219,-101.974,179.682,22.371,153.012
C04265=1099.471,438.972,-101.931,179.679,22.359,153.010
C04266=1099.465,438.726,-101.889,179.677,22.347,153.007
C04267=1099.459,438.480,-101.847,179.676,22.336,153.004
C04268=1099.450,438.147,-101.789,179.673,22.320,153.001
C04269=1099.443,437.813,-101.732,179.670,22.304,152.997
C04270=1099.435,437.480,-101.675,179.667,22.289,152.994
C04271=1099.426,437.146,-101.618,179.665,22.274,152.990
C04272=1099.420,436.900,-101.576,179.662,22.262,152.988
C04273=1099.414,436.654,-101.534,179.660,22.251,152.985
C04274=1099.408,436.408,-101.491,179.658,22.240,152.983
C04275=1099.402,436.161,-101.450,179.656,22.228,152.980
C04276=1099.396,435.915,-101.407,179.653,22.217,152.978
C04277=1099.390,435.669,-101.365,179.652,22.206,152.975
C04278=1099.384,435.422,-101.323,179.649,22.195,152.973
C04279=1099.378,435.176,-101.281,179.648,22.184,152.970
C04280=1099.372,434.930,-101.239,179.645,22.173,152.968
C04281=1099.366,434.684,-101.198,179.644,22.162,152.965
C04282=1099.360,434.437,-101.155,179.641,22.151,152.963
C04283=1099.354,434.191,-101.113,179.639,22.140,152.961
C04284=1099.348,433.945,-101.072,179.637,22.129,152.958
C04285=1099.343,433.698,-101.030,179.634,22.118,152.956
C04286=1099.336,433.452,-100.987,179.633,22.108,152.953
C04287=1099.330,433.206,-100.946,179.630,22.097,152.951
C04288=1099.324,432.960,-100.904,179.628,22.086,152.949
C04289=1099.318,432.713,-100.863,179.626,22.075,152.946
C04290=1099.312,432.466,-100.821,179.624,22.065,152.944
C04291=1099.307,432.220,-100.779,179.621,22.054,152.942
C04292=1099.301,431.974,-100.737,179.620,22.044,152.939
C04293=1099.295,431.728,-100.696,179.618,22.034,152.937
C04294=1099.289,431.481,-100.655,179.615,22.023,152.935
C04295=1099.282,431.234,-100.613,179.613,22.013,152.932
C04296=1099.276,430.988,-100.571,179.611,22.002,152.930
C04297=1099.270,430.742,-100.530,179.609,21.992,152.928
C04298=1099.264,430.496,-100.488,179.606,21.981,152.926
C04299=1099.258,430.250,-100.447,179.604,21.972,152.924
C04300=1099.252,430.003,-100.405,179.602,21.961,152.921
C04301=1099.246,429.757,-100.364,179.600,21.951,152.919
C04302=1099.240,429.510,-100.323,179.598,21.941,152.917
C04303=1099.234,429.263,-100.281,179.595,21.930,152.915
C04304=1099.228,429.017,-100.240,179.593,21.920,152.912
C04305=1099.222,428.771,-100.198,179.591,21.910,152.910
C04306=1099.217,428.524,-100.158,179.588,21.900,152.908
C04307=1099.211,428.278,-100.116,179.586,21.891,152.906
C04308=1099.204,428.031,-100.074,179.584,21.881,152.904
C04309=1099.199,427.784,-100.034,179.581,21.871,152.902
C04310=1099.193,427.538,-99.992,179.579,21.861,152.900
C04311=1099.186,427.292,-99.951,179.578,21.851,152.897
C04312=1099.180,427.045,-99.911,179.575,21.842,152.895
C04313=1099.174,426.799,-99.869,179.572,21.832,152.893
C04314=1099.169,426.552,-99.828,179.571,21.822,152.891
C04315=1099.163,426.306,-99.787,179.568,21.812,152.889
C04316=1099.157,426.059,-99.746,179.566,21.803,152.887
C04317=1099.150,425.813,-99.705,179.563,21.793,152.885
C04318=1099.145,425.567,-99.665,179.561,21.783,152.883
C04319=1099.139,425.320,-99.623,179.559,21.774,152.881
C04320=1099.133,425.096,-99.585,179.557,21.765,152.879
C04321=1099.127,424.872,-99.549,179.554,21.756,152.877
C04322=1099.122,424.648,-99.512,179.553,21.748,152.875
C04323=1099.117,424.425,-99.475,179.551,21.739,152.874
C04324=1099.112,424.201,-99.437,179.549,21.731,152.872
C04325=1099.106,423.977,-99.401,179.546,21.722,152.870
C04326=1099.101,423.754,-99.364,179.544,21.713,152.868
C04327=1099.096,423.530,-99.326,179.543,21.705,152.866
C04328=1099.089,423.283,-99.286,179.540,21.696,152.865
C04329=1099.084,423.037,-99.246,179.537,21.686,152.862
C04330=1099.078,422.790,-99.204,179.535,21.677,152.861
C04331=1099.071,422.544,-99.164,179.533,21.668,152.859
C04332=1099.066,422.297,-99.123,179.531,21.659,152.857
C04333=1099.060,422.050,-99.082,179.528,21.650,152.855
C04334=1099.054,421.804,-99.042,179.526,21.641,152.853
C04335=1099.048,421.557,-99.002,179.524,21.632,152.851
C04336=1099.042,421.310,-98.961,179.522,21.623,152.849
C04337=1099.036,421.064,-98.920,179.519,21.614,152.847
C04338=1099.029,420.818,-98.880,179.516,21.604,152.845
C04339=1099.024,420.571,-98.839,179.514,21.595,152.844
C04340=1099.017,420.324,-98.799,179.511,21.587,152.842
C04341=1099.012,420.077,-98.758,179.509,21.577,152.840
C04342=1099.006,419.832,-98.718,179.507,21.569,152.838
C04343=1099.001,419.584,-98.678,179.504,21.560,152.836
C04344=1098.994,419.338,-98.638,179.502,21.551,152.834
C04345=1098.989,419.091,-98.598,179.500,21.542,152.833
C04346=1098.982,418.844,-98.557,179.497,21.534,152.831
C04347=1098.977,418.598,-98.517,179.495,21.525,152.829
C04348=1098.970,418.351,-98.476,179.492,21.516,152.827
C04349=1098.965,418.105,-98.436,179.490,21.508,152.826
C04350=1098.959,417.858,-98.397,179.488,21.499,152.824
C04351=1098.953,417.611,-98.357,179.485,21.490,152.822
C04352=1098.947,417.364,-98.316,179.483,21.482,152.820
C04353=1098.941,417.118,-98.276,179.480,21.473,152.818
C04354=1098.935,416.870,-98.236,179.478,21.464,152.817
C04355=1098.930,416.625,-98.196,179.476,21.456,152.815
C04356=1098.923,416.378,-98.156,179.473,21.447,152.813
C04357=1098.918,416.131,-98.116,179.471,21.440,152.812
C04358=1098.911,415.884,-98.075,179.469,21.431,152.810
C04359=1098.905,415.637,-98.036,179.466,21.423,152.808
C04360=1098.899,415.391,-97.996,179.464,21.415,152.807
C04361=1098.894,415.144,-97.956,179.461,21.406,152.805
C04362=1098.888,414.897,-97.916,179.459,21.398,152.803
C04363=1098.881,414.651,-97.876,179.456,21.389,152.802
C04364=1098.875,414.404,-97.837,179.454,21.381,152.800
C04365=1098.869,414.157,-97.796,179.452,21.373,152.798
C04366=1098.864,413.911,-97.757,179.449,21.365,152.797
C04367=1098.858,413.664,-97.717,179.447,21.357,152.795
C04368=1098.852,413.417,-97.677,179.444,21.349,152.793
C04369=1098.846,413.170,-97.638,179.441,21.341,152.792
C04370=1098.840,412.924,-97.598,179.439,21.332,152.790
C04371=1098.834,412.677,-97.558,179.437,21.325,152.789
C04372=1098.828,412.429,-97.519,179.434,21.317,152.787
C04373=1098.822,412.184,-97.479,179.432,21.309,152.785
C04374=1098.817,411.936,-97.439,179.429,21.300,152.784
C04375=1098.811,411.689,-97.400,179.427,21.293,152.782
C04376=1098.805,411.473,-97.365,179.424,21.286,152.781
C04377=1098.800,411.256,-97.331,179.422,21.279,152.780
C04378=1098.796,411.039,-97.296,179.420,21.272,152.778
C04379=1098.790,410.823,-97.261,179.418,21.265,152.777
C04380=1098.784,410.605,-97.226,179.416,21.258,152.775
C04381=1098.779,410.388,-97.192,179.414,21.251,152.774
C04382=1098.774,410.172,-97.157,179.412,21.244,152.773
C04383=1098.769,409.955,-97.122,179.409,21.237,152.771
C04384=1098.763,409.708,-97.083,179.408,21.230,152.770
C04385=1098.758,409.461,-97.044,179.405,21.222,152.768
C04386=1098.752,409.214,-97.004,179.402,21.214,152.767
C04387=1098.746,408.968,-96.965,179.399,21.206,152.765
C04388=1098.740,408.720,-96.926,179.397,21.199,152.764
C04389=1098.734,408.473,-96.886,179.395,21.191,152.762
C04390=1098.728,408.227,-96.847,179.392,21.184,152.761
C04391=1098.722,407.980,-96.808,179.390,21.176,152.759
C04392=1098.717,407.733,-96.769,179.387,21.169,152.758
C04393=1098.711,407.486,-96.729,179.385,21.162,152.757
C04394=1098.705,407.240,-96.690,179.382,21.154,152.755
C04395=1098.699,406.993,-96.651,179.379,21.146,152.754
C04396=1098.693,406.745,-96.612,179.378,21.139,152.752
C04397=1098.687,406.499,-96.573,179.375,21.132,152.751
C04398=1098.681,406.252,-96.534,179.373,21.124,152.749
C04399=1098.676,406.005,-96.495,179.370,21.117,152.748
C04400=1098.670,405.758,-96.456,179.367,21.109,152.747
C04401=1098.664,405.512,-96.417,179.365,21.102,152.745
C04402=1098.658,405.264,-96.377,179.362,21.094,152.744
C04403=1098.652,405.018,-96.339,179.360,21.088,152.742
C04404=1098.646,404.771,-96.300,179.357,21.080,152.741
C04405=1098.641,404.524,-96.261,179.355,21.073,152.740
C04406=1098.635,404.277,-96.222,179.352,21.066,152.738
C04407=1098.629,404.030,-96.184,179.350,21.059,152.737
C04408=1098.623,403.783,-96.145,179.347,21.052,152.736
C04409=1098.617,403.537,-96.105,179.345,21.045,152.734
C04410=1098.611,403.289,-96.067,179.342,21.037,152.733
C04411=1098.605,403.043,-96.028,179.340,21.030,152.732
C04412=1098.599,402.795,-95.990,179.337,21.023,152.730
C04413=1098.593,402.549,-95.951,179.335,21.016,152.729
C04414=1098.587,402.302,-95.912,179.332,21.009,152.728
C04415=1098.582,402.055,-95.873,179.329,21.002,152.726
C04416=1098.576,401.809,-95.835,179.327,20.995,152.725
C04417=1098.570,401.561,-95.796,179.324,20.988,152.724
C04418=1098.564,401.315,-95.758,179.321,20.981,152.723
C04419=1098.558,401.067,-95.719,179.319,20.974,152.721
C04420=1098.553,400.820,-95.681,179.317,20.968,152.720
C04421=1098.547,400.574,-95.642,179.314,20.961,152.719
C04422=1098.541,400.326,-95.603,179.312,20.954,152.717
C04423=1098.535,400.080,-95.565,179.309,20.947,152.716
C04424=1098.529,399.832,-95.526,179.306,20.940,152.715
C04425=1098.523,399.585,-95.488,179.304,20.934,152.714
C04426=1098.518,399.339,-95.449,179.301,20.927,152.712
C04427=1098.511,399.092,-95.411,179.299,20.920,152.711
C04428=1098.506,398.845,-95.373,179.296,20.913,152.710
C04429=1098.500,398.598,-95.335,179.293,20.907,152.709
C04430=1098.494,398.351,-95.296,179.291,20.900,152.708
C04431=1098.488,398.104,-95.258,179.288,20.893,152.706
C04432=1098.483,397.887,-95.224,179.286,20.888,152.705
C04433=1098.478,397.671,-95.191,179.284,20.882,152.704
C04434=1098.473,397.454,-95.157,179.281,20.876,152.703
C04435=1098.467,397.237,-95.124,179.279,20.871,152.702
C04436=1098.462,397.020,-95.090,179.277,20.865,152.701
C04437=1098.457,396.804,-95.056,179.274,20.859,152.700
C04438=1098.452,396.587,-95.023,179.273,20.853,152.699
C04439=1098.447,396.370,-94.989,179.270,20.848,152.698
C04440=1098.441,396.123,-94.951,179.268,20.841,152.697
C04441=1098.435,395.877,-94.914,179.265,20.834,152.696
C04442=1098.429,395.629,-94.875,179.262,20.828,152.695
C04443=1098.424,395.382,-94.837,179.260,20.822,152.693
C04444=1098.418,395.136,-94.799,179.257,20.815,152.692
C04445=1098.412,394.888,-94.761,179.254,20.809,152.691
C04446=1098.406,394.641,-94.723,179.252,20.803,152.690
C04447=1098.400,394.394,-94.685,179.249,20.796,152.689
C04448=1098.394,394.148,-94.647,179.246,20.790,152.688
C04449=1098.389,393.900,-94.609,179.244,20.783,152.687
C04450=1098.383,393.654,-94.571,179.241,20.777,152.686
C04451=1098.377,393.406,-94.533,179.239,20.771,152.684
C04452=1098.371,393.160,-94.496,179.236,20.764,152.683
C04453=1098.365,392.912,-94.458,179.233,20.758,152.682
C04454=1098.360,392.665,-94.420,179.231,20.752,152.681
C04455=1098.354,392.418,-94.382,179.228,20.746,152.680
C04456=1098.348,392.172,-94.345,179.225,20.740,152.679
C04457=1098.342,391.924,-94.306,179.222,20.734,152.678
C04458=1098.336,391.677,-94.269,179.220,20.728,152.677
C04459=1098.330,391.430,-94.232,179.217,20.722,152.676
C04460=1098.324,391.183,-94.194,179.215,20.716,152.675
C04461=1098.318,390.937,-94.156,179.211,20.710,152.674
C04462=1098.313,390.689,-94.119,179.209,20.703,152.673
C04463=1098.307,390.442,-94.081,179.207,20.697,152.672
C04464=1098.300,390.195,-94.043,179.204,20.692,152.671
C04465=1098.294,389.948,-94.006,179.201,20.686,152.670
C04466=1098.289,389.701,-93.968,179.198,20.679,152.669
C04467=1098.283,389.454,-93.931,179.195,20.674,152.668
C04468=1098.277,389.207,-93.894,179.193,20.667,152.667
C04469=1098.271,388.960,-93.856,179.190,20.662,152.666
C04470=1098.265,388.713,-93.818,179.188,20.656,152.665
C04471=1098.260,388.466,-93.781,179.185,20.650,152.664
C04472=1098.254,388.219,-93.743,179.182,20.644,152.663
C04473=1098.248,387.972,-93.706,179.179,20.638,152.662
C04474=1098.242,387.725,-93.669,179.177,20.632,152.661
C04475=1098.236,387.478,-93.632,179.174,20.627,152.660
C04476=1098.230,387.231,-93.594,179.171,20.621,152.659
C04477=1098.225,386.984,-93.557,179.169,20.615,152.658
C04478=1098.219,386.737,-93.520,179.165,20.609,152.657
C04479=1098.213,386.490,-93.483,179.162,20.603,152.656
C04480=1098.207,386.243,-93.445,179.160,20.598,152.655
C04481=1098.202,385.996,-93.408,179.157,20.592,152.654
C04482=1098.196,385.748,-93.371,179.155,20.586,152.653
C04483=1098.189,385.502,-93.334,179.152,20.580,152.652
C04484=1098.184,385.255,-93.296,179.149,20.575,152.651
C04485=1098.178,385.007,-93.259,179.147,20.569,152.650
C04486=1098.172,384.760,-93.222,179.144,20.564,152.650
C04487=1098.167,384.513,-93.185,179.141,20.558,152.649
C04488=1098.162,384.303,-93.154,179.138,20.553,152.648
C04489=1098.157,384.093,-93.122,179.136,20.548,152.647
C04490=1098.152,383.882,-93.090,179.134,20.544,152.646
C04491=1098.147,383.671,-93.059,179.131,20.538,152.646
C04492=1098.143,383.461,-93.027,179.129,20.534,152.645
C04493=1098.137,383.251,-92.996,179.127,20.529,152.644
C04494=1098.133,383.041,-92.964,179.124,20.524,152.643
C04495=1098.127,382.830,-92.933,179.122,20.519,152.642
C04496=1098.122,382.583,-92.896,179.119,20.514,152.642
C04497=1098.116,382.335,-92.859,179.117,20.509,152.641
C04498=1098.110,382.089,-92.822,179.114,20.503,152.640
C04499=1098.104,381.842,-92.785,179.111,20.498,152.639
C04500=1098.099,381.595,-92.748,179.108,20.492,152.638
C04501=1098.092,381.348,-92.712,179.105,20.487,152.637
C04502=1098.087,381.100,-92.675,179.103,20.481,152.637
C04503=1098.080,380.853,-92.638,179.100,20.476,152.636
C04504=1098.075,380.606,-92.601,179.097,20.471,152.635
C04505=1098.069,380.359,-92.565,179.094,20.466,152.634
C04506=1098.063,380.111,-92.528,179.091,20.460,152.633
C04507=1098.058,379.865,-92.491,179.089,20.455,152.632
C04508=1098.052,379.618,-92.454,179.086,20.450,152.632
C04509=1098.046,379.370,-92.417,179.083,20.444,152.631
C04510=1098.040,379.123,-92.381,179.080,20.439,152.630
C04511=1098.034,378.875,-92.345,179.077,20.434,152.629
C04512=1098.028,378.628,-92.308,179.075,20.428,152.628
C04513=1098.023,378.382,-92.272,179.072,20.423,152.628
C04514=1098.017,378.135,-92.235,179.069,20.418,152.627
C04515=1098.011,377.887,-92.198,179.066,20.413,152.626
C04516=1098.005,377.640,-92.162,179.063,20.407,152.625
C04517=1098.000,377.393,-92.126,179.060,20.402,152.624
C04518=1097.994,377.146,-92.089,179.057,20.397,152.624
C04519=1097.988,376.898,-92.052,179.055,20.392,152.623
C04520=1097.982,376.651,-92.016,179.052,20.386,152.622
C04521=1097.977,376.403,-91.979,179.049,20.381,152.621
C04522=1097.971,376.157,-91.943,179.046,20.376,152.621
C04523=1097.965,375.910,-91.906,179.043,20.371,152.620
C04524=1097.959,375.662,-91.871,179.040,20.366,152.619
C04525=1097.954,375.415,-91.834,179.038,20.361,152.618
C04526=1097.948,375.168,-91.797,179.035,20.356,152.618
C04527=1097.942,374.921,-91.762,179.032,20.351,152.617
C04528=1097.936,374.673,-91.725,179.029,20.346,152.616
C04529=1097.931,374.426,-91.689,179.026,20.341,152.615
C04530=1097.924,374.179,-91.653,179.023,20.336,152.615
C04531=1097.919,373.931,-91.616,179.020,20.331,152.614
C04532=1097.913,373.685,-91.580,179.017,20.326,152.613
C04533=1097.907,373.437,-91.545,179.015,20.321,152.612
C04534=1097.901,373.190,-91.508,179.012,20.316,152.612
C04535=1097.896,372.942,-91.472,179.009,20.311,152.611
C04536=1097.890,372.696,-91.436,179.006,20.307,152.610
C04537=1097.884,372.448,-91.400,179.003,20.302,152.610
C04538=1097.878,372.201,-91.364,179.001,20.296,152.609
C04539=1097.873,371.954,-91.328,178.997,20.291,152.608
C04540=1097.867,371.706,-91.292,178.994,20.287,152.608
C04541=1097.861,371.459,-91.256,178.991,20.282,152.607
C04542=1097.855,371.212,-91.220,178.989,20.277,152.606
C04543=1097.849,370.964,-91.184,178.986,20.272,152.606
C04544=1097.840,370.571,-91.127,178.981,20.265,152.605
C04545=1097.831,370.178,-91.070,178.976,20.257,152.604
C04546=1097.822,369.783,-91.013,178.972,20.250,152.602
C04547=1097.812,369.390,-90.956,178.967,20.242,152.602
C04548=1097.807,369.143,-90.920,178.964,20.237,152.601
C04549=1097.801,368.895,-90.884,178.961,20.232,152.600
C04550=1097.796,368.648,-90.848,178.958,20.227,152.600
C04551=1097.790,368.401,-90.812,178.956,20.223,152.599
C04552=1097.784,368.154,-90.777,178.953,20.218,152.598
C04553=1097.778,367.906,-90.741,178.950,20.214,152.598
C04554=1097.772,367.658,-90.705,178.947,20.209,152.597
C04555=1097.767,367.411,-90.670,178.944,20.204,152.596
C04556=1097.761,367.164,-90.634,178.942,20.200,152.596
C04557=1097.755,366.917,-90.599,178.938,20.195,152.595
C04558=1097.749,366.669,-90.563,178.935,20.190,152.595
C04559=1097.744,366.422,-90.528,178.932,20.185,152.594
C04560=1097.738,366.174,-90.492,178.930,20.181,152.593
C04561=1097.732,365.927,-90.457,178.927,20.177,152.593
C04562=1097.726,365.680,-90.421,178.924,20.172,152.592
C04563=1097.721,365.433,-90.385,178.921,20.167,152.591
C04564=1097.715,365.185,-90.350,178.917,20.163,152.591
C04565=1097.709,364.937,-90.314,178.915,20.158,152.590
C04566=1097.703,364.690,-90.279,178.912,20.154,152.590
C04567=1097.697,364.443,-90.243,178.909,20.149,152.589
C04568=1097.692,364.196,-90.208,178.906,20.145,152.589
C04569=1097.686,363.948,-90.172,178.903,20.141,152.588
C04570=1097.681,363.701,-90.137,178.900,20.136,152.588
C04571=1097.674,363.453,-90.102,178.897,20.132,152.587
C04572=1097.669,363.206,-90.067,178.895,20.127,152.586
C04573=1097.663,362.959,-90.031,178.891,20.123,152.586
C04574=1097.657,362.711,-89.996,178.888,20.118,152.585
C04575=1097.651,362.463,-89.961,178.885,20.114,152.585
C04576=1097.646,362.216,-89.925,178.883,20.110,152.584
C04577=1097.639,361.969,-89.890,178.880,20.105,152.584
C04578=1097.634,361.721,-89.855,178.876,20.101,152.583
C04579=1097.629,361.474,-89.820,178.873,20.096,152.583
C04580=1097.623,361.227,-89.784,178.871,20.092,152.582
C04581=1097.617,360.979,-89.750,178.867,20.088,152.582
C04582=1097.611,360.732,-89.715,178.864,20.083,152.581
C04583=1097.605,360.485,-89.679,178.862,20.079,152.580
C04584=1097.600,360.236,-89.644,178.859,20.075,152.580
C04585=1097.594,359.989,-89.609,178.855,20.070,152.579
C04586=1097.588,359.742,-89.575,178.853,20.067,152.579
C04587=1097.582,359.495,-89.539,178.850,20.062,152.578
C04588=1097.577,359.247,-89.504,178.846,20.058,152.578
C04589=1097.570,359.000,-89.469,178.844,20.054,152.577
C04590=1097.565,358.752,-89.435,178.841,20.050,152.577
C04591=1097.558,358.505,-89.399,178.837,20.045,152.576
C04592=1097.553,358.257,-89.365,178.835,20.041,152.576
C04593=1097.548,358.010,-89.329,178.831,20.037,152.576
C04594=1097.541,357.762,-89.295,178.828,20.033,152.575
C04595=1097.536,357.515,-89.260,178.826,20.029,152.575
C04596=1097.528,357.136,-89.207,178.820,20.022,152.574
C04597=1097.518,356.757,-89.154,178.816,20.016,152.573
C04598=1097.510,356.379,-89.100,178.812,20.009,152.572
C04599=1097.501,356.000,-89.047,178.807,20.003,152.572
C04600=1097.495,355.753,-89.013,178.804,19.999,152.571
C04601=1097.489,355.505,-88.978,178.801,19.995,152.571
C04602=1097.483,355.258,-88.943,178.798,19.991,152.570
C04603=1097.478,355.011,-88.908,178.795,19.987,152.570
C04604=1097.472,354.764,-88.874,178.792,19.983,152.569
C04605=1097.466,354.515,-88.839,178.789,19.978,152.569
C04606=1097.461,354.268,-88.805,178.786,19.975,152.568
C04607=1097.455,354.020,-88.770,178.783,19.970,152.568
C04608=1097.449,353.772,-88.736,178.780,19.967,152.568
C04609=1097.444,353.525,-88.701,178.777,19.963,152.567
C04610=1097.438,353.278,-88.666,178.774,19.958,152.567
C04611=1097.433,353.031,-88.632,178.771,19.955,152.566
C04612=1097.426,352.783,-88.597,178.767,19.951,152.566
C04613=1097.421,352.535,-88.563,178.765,19.947,152.565
C04614=1097.415,352.288,-88.529,178.762,19.943,152.565
C04615=1097.409,352.040,-88.494,178.758,19.939,152.565
C04616=1097.404,351.792,-88.460,178.756,19.935,152.564
C04617=1097.398,351.545,-88.426,178.752,19.931,152.564
C04618=1097.392,351.298,-88.392,178.750,19.927,152.563
C04619=1097.386,351.049,-88.357,178.746,19.923,152.563
C04620=1097.380,350.802,-88.322,178.744,19.920,152.563
C04621=1097.374,350.555,-88.288,178.740,19.916,152.562
C04622=1097.369,350.307,-88.254,178.738,19.912,152.562
C04623=1097.363,350.059,-88.219,178.734,19.908,152.561
C04624=1097.357,349.812,-88.185,178.731,19.904,152.561
C04625=1097.352,349.564,-88.151,178.728,19.900,152.561
C04626=1097.346,349.317,-88.117,178.725,19.896,152.560
C04627=1097.340,349.069,-88.083,178.722,19.892,152.560
C04628=1097.335,348.822,-88.049,178.719,19.888,152.560
C04629=1097.329,348.573,-88.014,178.716,19.885,152.559
C04630=1097.323,348.326,-87.980,178.713,19.881,152.559
C04631=1097.317,348.079,-87.946,178.710,19.877,152.558
C04632=1097.312,347.831,-87.913,178.707,19.873,152.558
C04633=1097.306,347.583,-87.878,178.704,19.870,152.558
C04634=1097.301,347.336,-87.844,178.701,19.866,152.557
C04635=1097.294,347.088,-87.810,178.698,19.862,152.557
C04636=1097.289,346.840,-87.776,178.695,19.858,152.557
C04637=1097.283,346.593,-87.742,178.691,19.855,152.556
C04638=1097.278,346.345,-87.708,178.688,19.851,152.556
C04639=1097.272,346.097,-87.674,178.685,19.847,152.556
C04640=1097.266,345.850,-87.640,178.682,19.843,152.555
C04641=1097.260,345.603,-87.606,178.679,19.839,152.555
C04642=1097.255,345.355,-87.573,178.676,19.836,152.554
C04643=1097.248,345.107,-87.538,178.672,19.832,152.554
C04644=1097.243,344.859,-87.505,178.670,19.829,152.554
C04645=1097.237,344.612,-87.471,178.667,19.825,152.553
C04646=1097.231,344.365,-87.437,178.664,19.822,152.553
C04647=1097.225,344.117,-87.404,178.661,19.818,152.553
C04648=1097.217,343.740,-87.352,178.656,19.812,152.552
C04649=1097.208,343.364,-87.300,178.651,19.807,152.552
C04650=1097.200,342.988,-87.250,178.646,19.801,152.551
C04651=1097.191,342.612,-87.198,178.641,19.796,152.551
C04652=1097.185,342.364,-87.164,178.639,19.793,152.551
C04653=1097.180,342.116,-87.131,178.636,19.789,152.550
C04654=1097.174,341.869,-87.098,178.632,19.785,152.550
C04655=1097.168,341.622,-87.064,178.630,19.782,152.550
C04656=1097.162,341.374,-87.031,178.626,19.778,152.549
C04657=1097.157,341.126,-86.997,178.623,19.775,152.549
C04658=1097.151,340.878,-86.963,178.620,19.771,152.549
C04659=1097.145,340.631,-86.930,178.617,19.768,152.549
C04660=1097.140,340.383,-86.897,178.614,19.764,152.548
C04661=1097.134,340.135,-86.863,178.611,19.760,152.548
C04662=1097.128,339.887,-86.829,178.608,19.757,152.548
C04663=1097.123,339.640,-86.796,178.605,19.753,152.547
C04664=1097.117,339.392,-86.763,178.602,19.750,152.547
C04665=1097.111,339.144,-86.729,178.598,19.747,152.547
C04666=1097.106,338.896,-86.695,178.596,19.743,152.546
C04667=1097.099,338.649,-86.663,178.592,19.739,152.546
C04668=1097.094,338.401,-86.629,178.589,19.736,152.546
C04669=1097.088,338.153,-86.596,178.586,19.733,152.546
C04670=1097.083,337.905,-86.563,178.583,19.729,152.545
C04671=1097.077,337.658,-86.528,178.580,19.726,152.545
C04672=1097.071,337.410,-86.496,178.577,19.723,152.545
C04673=1097.065,337.162,-86.462,178.573,19.719,152.545
C04674=1097.059,336.914,-86.429,178.571,19.716,152.544
C04675=1097.054,336.667,-86.396,178.567,19.712,152.544
C04676=1097.048,336.419,-86.363,178.564,19.709,152.544
C04677=1097.042,336.171,-86.330,178.561,19.706,152.544
C04678=1097.036,335.923,-86.296,178.558,19.702,152.543
C04679=1097.030,335.676,-86.264,178.555,19.699,152.543
C04680=1097.025,335.428,-86.230,178.551,19.696,152.543
C04681=1097.020,335.180,-86.197,178.548,19.693,152.543
C04682=1097.013,334.933,-86.165,178.546,19.689,152.542
C04683=1097.008,334.685,-86.131,178.542,19.686,152.542
C04684=1097.002,334.437,-86.098,178.539,19.682,152.542
C04685=1096.996,334.189,-86.065,178.536,19.679,152.542
C04686=1096.990,333.942,-86.032,178.533,19.676,152.542
C04687=1096.985,333.693,-85.999,178.530,19.673,152.541
C04688=1096.979,333.446,-85.967,178.527,19.670,152.541
C04689=1096.974,333.198,-85.933,178.523,19.666,152.541
C04690=1096.968,332.950,-85.900,178.521,19.663,152.541
C04691=1096.962,332.703,-85.867,178.518,19.660,152.540
C04692=1096.957,332.455,-85.834,178.514,19.656,152.540
C04693=1096.951,332.206,-85.801,178.511,19.653,152.540
C04694=1096.946,331.959,-85.769,178.508,19.650,152.540
C04695=1096.939,331.712,-85.736,178.505,19.647,152.540
C04696=1096.934,331.464,-85.703,178.502,19.644,152.539
C04697=1096.928,331.216,-85.671,178.499,19.641,152.539
C04698=1096.922,330.968,-85.638,178.495,19.637,152.539
C04699=1096.916,330.720,-85.605,178.492,19.634,152.539
C04700=1096.907,330.338,-85.554,178.487,19.629,152.539
C04701=1096.898,329.956,-85.504,178.483,19.625,152.538
C04702=1096.889,329.573,-85.454,178.477,19.620,152.538
C04703=1096.880,329.192,-85.403,178.473,19.615,152.538
C04704=1096.874,328.944,-85.371,178.469,19.612,152.538
C04705=1096.869,328.696,-85.338,178.466,19.609,152.537
C04706=1096.863,328.447,-85.306,178.464,19.606,152.537
C04707=1096.856,328.200,-85.273,178.460,19.602,152.537
C04708=1096.852,327.952,-85.241,178.457,19.599,152.537
C04709=1096.845,327.704,-85.208,178.454,19.597,152.537
C04710=1096.840,327.456,-85.176,178.451,19.594,152.537
C04711=1096.834,327.208,-85.143,178.447,19.590,152.536
C04712=1096.829,326.961,-85.111,178.444,19.587,152.536
C04713=1096.822,326.713,-85.079,178.441,19.584,152.536
C04714=1096.817,326.465,-85.046,178.438,19.582,152.536
C04715=1096.811,326.217,-85.013,178.435,19.578,152.536
C04716=1096.805,325.970,-84.982,178.432,19.575,152.536
C04717=1096.799,325.722,-84.949,178.429,19.572,152.535
C04718=1096.794,325.474,-84.916,178.426,19.570,152.535
C04719=1096.788,325.226,-84.885,178.422,19.566,152.535
C04720=1096.782,324.978,-84.852,178.419,19.563,152.535
C04721=1096.776,324.730,-84.820,178.416,19.560,152.535
C04722=1096.771,324.482,-84.787,178.413,19.558,152.535
C04723=1096.765,324.235,-84.755,178.409,19.554,152.535
C04724=1096.759,323.987,-84.723,178.406,19.551,152.534
C04725=1096.754,323.739,-84.691,178.404,19.548,152.534
C04726=1096.748,323.491,-84.659,178.400,19.546,152.534
C04727=1096.742,323.243,-84.626,178.397,19.542,152.534
C04728=1096.737,322.995,-84.594,178.394,19.539,152.534
C04729=1096.731,322.747,-84.562,178.391,19.536,152.534
C04730=1096.725,322.499,-84.530,178.388,19.533,152.534
C04731=1096.720,322.251,-84.498,178.385,19.531,152.533
C04732=1096.714,322.004,-84.465,178.381,19.527,152.533
C04733=1096.709,321.756,-84.433,178.378,19.525,152.533
C04734=1096.703,321.508,-84.401,178.375,19.521,152.533
C04735=1096.697,321.260,-84.370,178.372,19.519,152.533
C04736=1096.691,321.012,-84.338,178.369,19.516,152.533
C04737=1096.685,320.764,-84.306,178.365,19.512,152.533
C04738=1096.681,320.516,-84.273,178.362,19.510,152.533
C04739=1096.675,320.268,-84.241,178.359,19.507,152.532
C04740=1096.669,320.020,-84.210,178.356,19.504,152.532
C04741=1096.663,319.773,-84.177,178.353,19.501,152.532
C04742=1096.658,319.525,-84.145,178.349,19.498,152.532
C04743=1096.652,319.277,-84.113,178.347,19.495,152.532
C04744=1096.646,319.030,-84.082,178.344,19.492,152.532
C04745=1096.640,318.781,-84.050,178.341,19.490,152.532
C04746=1096.635,318.533,-84.019,178.338,19.487,152.531
C04747=1096.629,318.285,-83.987,178.334,19.484,152.531
C04748=1096.624,318.037,-83.954,178.331,19.481,152.531
C04749=1096.619,317.789,-83.922,178.328,19.478,152.531
C04750=1096.613,317.541,-83.891,178.325,19.475,152.531
C04751=1096.607,317.293,-83.859,178.322,19.472,152.531
C04752=1096.599,316.904,-83.809,178.316,19.468,152.531
C04753=1096.590,316.515,-83.759,178.312,19.464,152.531
C04754=1096.581,316.126,-83.710,178.307,19.459,152.530
C04755=1096.572,315.736,-83.660,178.302,19.455,152.530
C04756=1096.567,315.489,-83.628,178.298,19.451,152.530
C04757=1096.561,315.241,-83.596,178.295,19.449,152.530
C04758=1096.555,314.993,-83.564,178.292,19.446,152.530
C04759=1096.550,314.745,-83.534,178.289,19.443,152.530
C04760=1096.544,314.497,-83.502,178.286,19.441,152.530
C04761=1096.538,314.249,-83.470,178.283,19.438,152.530
C04762=1096.532,314.001,-83.438,178.280,19.435,152.530
C04763=1096.526,313.753,-83.408,178.276,19.432,152.530
C04764=1096.520,313.505,-83.376,178.273,19.430,152.530
C04765=1096.515,313.258,-83.344,178.270,19.427,152.530
C04766=1096.509,313.009,-83.314,178.267,19.425,152.530
C04767=1096.503,312.762,-83.282,178.264,19.422,152.530
C04768=1096.497,312.513,-83.250,178.260,19.419,152.529
C04769=1096.491,312.266,-83.220,178.257,19.417,152.529
C04770=1096.486,312.018,-83.188,178.254,19.414,152.529
C04771=1096.480,311.770,-83.157,178.251,19.412,152.529
C04772=1096.474,311.522,-83.126,178.247,19.409,152.529
C04773=1096.469,311.273,-83.094,178.244,19.406,152.529
C04774=1096.462,311.026,-83.063,178.241,19.403,152.529
C04775=1096.457,310.779,-83.031,178.238,19.401,152.529
C04776=1096.451,310.530,-83.000,178.235,19.398,152.529
C04777=1096.445,310.283,-82.969,178.232,19.396,152.529
C04778=1096.440,310.034,-82.938,178.229,19.393,152.529
C04779=1096.433,309.786,-82.907,178.225,19.390,152.529
C04780=1096.428,309.538,-82.876,178.222,19.388,152.529
C04781=1096.423,309.289,-82.844,178.218,19.385,152.529
C04782=1096.417,309.042,-82.813,178.215,19.382,152.529
C04783=1096.411,308.794,-82.782,178.212,19.380,152.529
C04784=1096.405,308.547,-82.751,178.209,19.378,152.529
C04785=1096.400,308.298,-82.720,178.206,19.375,152.529
C04786=1096.394,308.050,-82.690,178.203,19.372,152.529
C04787=1096.388,307.803,-82.658,178.200,19.370,152.529
C04788=1096.382,307.554,-82.627,178.196,19.367,152.529
C04789=1096.377,307.306,-82.596,178.193,19.365,152.529
C04790=1096.371,307.059,-82.565,178.190,19.362,152.529
C04791=1096.366,306.811,-82.534,178.187,19.359,152.529
C04792=1096.359,306.562,-82.504,178.183,19.357,152.529
C04793=1096.354,306.315,-82.472,178.180,19.354,152.529
C04794=1096.348,306.067,-82.442,178.177,19.351,152.528
C04795=1096.343,305.819,-82.411,178.174,19.349,152.529
C04796=1096.337,305.571,-82.380,178.170,19.346,152.528
C04797=1096.331,305.323,-82.348,178.167,19.344,152.528
C04798=1096.325,305.075,-82.318,178.164,19.342,152.528
C04799=1096.320,304.827,-82.287,178.161,19.339,152.528
C04800=1096.315,304.579,-82.257,178.158,19.336,152.528
C04801=1096.309,304.331,-82.226,178.155,19.334,152.528
C04802=1096.303,304.082,-82.195,178.152,19.331,152.528
C04803=1096.298,303.835,-82.163,178.149,19.329,152.528
C04804=1096.289,303.448,-82.116,178.143,19.324,152.528
C04805=1096.280,303.061,-82.068,178.138,19.321,152.528
C04806=1096.271,302.675,-82.020,178.134,19.317,152.528
C04807=1096.262,302.288,-81.972,178.128,19.313,152.528
C04808=1096.257,302.040,-81.942,178.125,19.310,152.528
C04809=1096.252,301.792,-81.911,178.122,19.308,152.528
C04810=1096.246,301.544,-81.881,178.118,19.305,152.528
C04811=1096.240,301.297,-81.850,178.115,19.303,152.528
C04812=1096.235,301.048,-81.819,178.112,19.300,152.528
C04813=1096.229,300.801,-81.789,178.109,19.298,152.528
C04814=1096.224,300.552,-81.758,178.106,19.295,152.528
C04815=1096.218,300.305,-81.728,178.103,19.293,152.528
C04816=1096.213,300.056,-81.698,178.100,19.290,152.528
C04817=1096.208,299.808,-81.667,178.096,19.288,152.528
C04818=1096.202,299.560,-81.637,178.093,19.285,152.528
C04819=1096.196,299.312,-81.606,178.090,19.283,152.528
C04820=1096.191,299.064,-81.575,178.087,19.281,152.528
C04821=1096.185,298.817,-81.545,178.084,19.278,152.528
C04822=1096.179,298.569,-81.515,178.080,19.276,152.528
C04823=1096.174,298.320,-81.485,178.077,19.273,152.528
C04824=1096.169,298.072,-81.454,178.074,19.271,152.528
C04825=1096.162,297.824,-81.423,178.071,19.268,152.528
C04826=1096.156,297.576,-81.393,178.068,19.266,152.528
C04827=1096.151,297.327,-81.364,178.064,19.264,152.528
C04828=1096.145,297.079,-81.333,178.061,19.261,152.528
C04829=1096.139,296.832,-81.303,178.058,19.259,152.528
C04830=1096.134,296.584,-81.272,178.055,19.257,152.528
C04831=1096.129,296.335,-81.242,178.052,19.254,152.528
C04832=1096.123,296.087,-81.212,178.048,19.252,152.528
C04833=1096.117,295.839,-81.182,178.045,19.250,152.528
C04834=1096.112,295.591,-81.152,178.042,19.247,152.528
C04835=1096.106,295.343,-81.122,178.039,19.245,152.528
C04836=1096.100,295.095,-81.092,178.035,19.243,152.529
C04837=1096.094,294.847,-81.062,178.032,19.240,152.528
C04838=1096.089,294.599,-81.031,178.029,19.238,152.529
C04839=1096.083,294.351,-81.002,178.026,19.235,152.529
C04840=1096.077,294.103,-80.971,178.022,19.233,152.529
C04841=1096.072,293.854,-80.942,178.019,19.231,152.529
C04842=1096.066,293.607,-80.911,178.016,19.228,152.529
C04843=1096.060,293.358,-80.882,178.013,19.226,152.529
C04844=1096.055,293.110,-80.851,178.010,19.223,152.529
C04845=1096.049,292.862,-80.822,178.006,19.221,152.529
C04846=1096.043,292.614,-80.791,178.003,19.219,152.529
C04847=1096.038,292.366,-80.762,178.000,19.217,152.529
C04848=1096.032,292.118,-80.731,177.997,19.214,152.529
C04849=1096.026,291.869,-80.702,177.993,19.212,152.529
C04850=1096.021,291.622,-80.671,177.990,19.210,152.529
C04851=1096.016,291.374,-80.642,177.987,19.208,152.529
C04852=1096.009,291.126,-80.613,177.984,19.205,152.529
C04853=1096.004,290.878,-80.583,177.980,19.203,152.529
C04854=1095.998,290.629,-80.553,177.977,19.200,152.529
C04855=1095.993,290.381,-80.523,177.975,19.199,152.529
C04856=1095.984,290.008,-80.478,177.970,19.195,152.529
C04857=1095.975,289.636,-80.433,177.965,19.192,152.530
C04858=1095.967,289.263,-80.389,177.960,19.188,152.530
C04859=1095.959,288.890,-80.344,177.955,19.185,152.530
C04860=1095.953,288.642,-80.315,177.952,19.183,152.530
C04861=1095.947,288.394,-80.285,177.949,19.181,152.530
C04862=1095.941,288.146,-80.255,177.945,19.178,152.530
C04863=1095.936,287.897,-80.226,177.942,19.176,152.530
C04864=1095.930,287.649,-80.196,177.939,19.174,152.530
C04865=1095.924,287.401,-80.167,177.935,19.172,152.530
C04866=1095.919,287.154,-80.137,177.932,19.170,152.530
C04867=1095.913,286.905,-80.108,177.930,19.168,152.530
C04868=1095.907,286.657,-80.078,177.926,19.166,152.530
C04869=1095.901,286.409,-80.049,177.923,19.163,152.531
C04870=1095.896,286.160,-80.019,177.920,19.161,152.531
C04871=1095.890,285.913,-79.991,177.916,19.159,152.531
C04872=1095.885,285.664,-79.961,177.913,19.157,152.531
C04873=1095.879,285.416,-79.931,177.910,19.155,152.531
C04874=1095.874,285.167,-79.902,177.906,19.152,152.531
C04875=1095.867,284.919,-79.873,177.903,19.150,152.531
C04876=1095.862,284.671,-79.843,177.900,19.147,152.531
C04877=1095.857,284.423,-79.814,177.897,19.145,152.531
C04878=1095.851,284.175,-79.785,177.894,19.144,152.531
C04879=1095.845,283.927,-79.755,177.891,19.141,152.531
C04880=1095.839,283.678,-79.726,177.888,19.139,152.531
C04881=1095.834,283.431,-79.697,177.884,19.137,152.531
C04882=1095.828,283.182,-79.667,177.881,19.135,152.531
C04883=1095.822,282.934,-79.638,177.878,19.133,152.532
C04884=1095.817,282.686,-79.608,177.874,19.130,152.532
C04885=1095.812,282.438,-79.579,177.871,19.128,152.532
C04886=1095.806,282.190,-79.550,177.868,19.126,152.532
C04887=1095.800,281.941,-79.520,177.865,19.124,152.532
C04888=1095.794,281.693,-79.492,177.862,19.122,152.532
C04889=1095.789,281.445,-79.463,177.859,19.120,152.532
C04890=1095.783,281.197,-79.434,177.855,19.118,152.532
C04891=1095.777,280.948,-79.404,177.852,19.115,152.532
C04892=1095.772,280.701,-79.375,177.849,19.114,152.532
C04893=1095.767,280.452,-79.347,177.845,19.111,152.533
C04894=1095.760,280.204,-79.318,177.842,19.109,152.533
C04895=1095.755,279.955,-79.288,177.840,19.108,152.533
C04896=1095.749,279.708,-79.259,177.836,19.105,152.533
C04897=1095.744,279.459,-79.230,177.833,19.103,152.533
C04898=1095.738,279.211,-79.201,177.830,19.101,152.533
C04899=1095.733,278.963,-79.172,177.826,19.099,152.533
C04900=1095.727,278.715,-79.143,177.823,19.097,152.533
C04901=1095.721,278.466,-79.115,177.819,19.095,152.533
C04902=1095.715,278.218,-79.085,177.817,19.093,152.533
C04903=1095.709,277.970,-79.056,177.814,19.091,152.534
C04904=1095.704,277.721,-79.027,177.810,19.089,152.534
C04905=1095.698,277.473,-78.998,177.807,19.086,152.534
C04906=1095.693,277.225,-78.970,177.804,19.084,152.534
C04907=1095.687,276.976,-78.941,177.800,19.082,152.534
C04908=1095.678,276.613,-78.899,177.796,19.080,152.534
C04909=1095.670,276.250,-78.857,177.791,19.076,152.534
C04910=1095.662,275.886,-78.814,177.787,19.074,152.534
C04911=1095.654,275.523,-78.773,177.782,19.071,152.535
C04912=1095.649,275.275,-78.744,177.779,19.069,152.535
C04913=1095.643,275.027,-78.715,177.775,19.066,152.535
C04914=1095.637,274.778,-78.687,177.772,19.064,152.535
C04915=1095.632,274.530,-78.658,177.769,19.062,152.535
C04916=1095.626,274.282,-78.629,177.766,19.061,152.535
C04917=1095.621,274.034,-78.601,177.763,19.058,152.535
C04918=1095.614,273.786,-78.572,177.759,19.056,152.535
C04919=1095.609,273.536,-78.543,177.756,19.054,152.536
C04920=1095.603,273.289,-78.514,177.754,19.052,152.536
C04921=1095.597,273.040,-78.486,177.750,19.051,152.536
C04922=1095.592,272.792,-78.458,177.747,19.048,152.536
C04923=1095.586,272.544,-78.429,177.743,19.046,152.536
C04924=1095.581,272.296,-78.401,177.740,19.044,152.536
C04925=1095.575,272.047,-78.372,177.737,19.042,152.536
C04926=1095.569,271.798,-78.344,177.734,19.041,152.536
C04927=1095.564,271.551,-78.315,177.731,19.038,152.537
C04928=1095.558,271.302,-78.287,177.727,19.037,152.537
C04929=1095.552,271.054,-78.259,177.724,19.034,152.537
C04930=1095.546,270.806,-78.230,177.721,19.032,152.537
C04931=1095.541,270.558,-78.202,177.718,19.031,152.537
C04932=1095.536,270.309,-78.173,177.715,19.029,152.537
C04933=1095.530,270.061,-78.145,177.711,19.027,152.537
C04934=1095.524,269.812,-78.117,177.708,19.024,152.537
C04935=1095.519,269.565,-78.088,177.704,19.023,152.538
C04936=1095.513,269.316,-78.060,177.702,19.021,152.538
C04937=1095.507,269.068,-78.032,177.699,19.019,152.538
C04938=1095.502,268.819,-78.003,177.695,19.017,152.538
C04939=1095.496,268.571,-77.975,177.692,19.015,152.538
C04940=1095.490,268.322,-77.947,177.689,19.014,152.538
C04941=1095.485,268.074,-77.919,177.686,19.011,152.539
C04942=1095.479,267.825,-77.891,177.682,19.009,152.539
C04943=1095.474,267.577,-77.863,177.679,19.007,152.539
C04944=1095.468,267.329,-77.835,177.676,19.005,152.539
C04945=1095.462,267.081,-77.807,177.673,19.003,152.539
C04946=1095.456,266.832,-77.778,177.670,19.002,152.539
C04947=1095.451,266.584,-77.750,177.666,18.999,152.539
C04948=1095.445,266.335,-77.722,177.663,18.997,152.539
C04949=1095.440,266.087,-77.694,177.660,18.996,152.540
C04950=1095.434,265.839,-77.666,177.657,18.994,152.540
C04951=1095.428,265.590,-77.638,177.653,18.992,152.540
C04952=1095.423,265.342,-77.610,177.650,18.990,152.540
C04953=1095.417,265.093,-77.581,177.648,18.988,152.540
C04954=1095.412,264.845,-77.554,177.644,18.986,152.540
C04955=1095.406,264.596,-77.525,177.641,18.984,152.541
C04956=1095.400,264.349,-77.498,177.637,18.982,152.541
C04957=1095.394,264.101,-77.470,177.635,18.981,152.541
C04958=1095.389,263.852,-77.442,177.631,18.979,152.541
C04959=1095.383,263.603,-77.414,177.628,18.977,152.541
C04960=1095.374,263.243,-77.374,177.624,18.975,152.541
C04961=1095.366,262.883,-77.333,177.618,18.972,152.542
C04962=1095.358,262.521,-77.293,177.614,18.969,152.542
C04963=1095.349,262.161,-77.253,177.609,18.966,152.542
C04964=1095.343,261.912,-77.225,177.606,18.965,152.542
C04965=1095.338,261.664,-77.197,177.603,18.963,152.542
C04966=1095.332,261.417,-77.169,177.599,18.961,152.543
C04967=1095.326,261.167,-77.142,177.596,18.959,152.543
C04968=1095.321,260.919,-77.114,177.593,18.957,152.543
C04969=1095.314,260.671,-77.086,177.590,18.955,152.543
C04970=1095.309,260.422,-77.059,177.587,18.954,152.543
C04971=1095.304,260.174,-77.031,177.583,18.952,152.544
C04972=1095.297,259.926,-77.003,177.581,18.950,152.544
C04973=1095.292,259.677,-76.976,177.577,18.948,152.544
C04974=1095.287,259.429,-76.948,177.574,18.946,152.544
C04975=1095.280,259.180,-76.921,177.571,18.945,152.544
C04976=1095.275,258.932,-76.893,177.568,18.943,152.544
C04977=1095.270,258.684,-76.865,177.564,18.941,152.545
C04978=1095.263,258.435,-76.838,177.561,18.939,152.545
C04979=1095.258,258.187,-76.810,177.558,18.938,152.545
C04980=1095.252,257.938,-76.783,177.555,18.935,152.545
C04981=1095.246,257.690,-76.755,177.551,18.934,152.545
C04982=1095.241,257.441,-76.728,177.549,18.932,152.545
C04983=1095.235,257.193,-76.700,177.545,18.930,152.546
C04984=1095.230,256.944,-76.673,177.542,18.928,152.546
C04985=1095.224,256.696,-76.646,177.538,18.926,152.546
C04986=1095.219,256.447,-76.618,177.536,18.925,152.546
C04987=1095.212,256.200,-76.591,177.532,18.923,152.546
C04988=1095.207,255.951,-76.564,177.529,18.921,152.547
C04989=1095.201,255.702,-76.535,177.526,18.919,152.547
C04990=1095.196,255.454,-76.509,177.523,18.918,152.547
C04991=1095.191,255.205,-76.481,177.519,18.915,152.547
C04992=1095.185,254.957,-76.454,177.517,18.914,152.547
C04993=1095.179,254.708,-76.426,177.513,18.912,152.547
C04994=1095.173,254.460,-76.400,177.510,18.910,152.548
C04995=1095.168,254.212,-76.372,177.507,18.909,152.548
C04996=1095.162,253.963,-76.345,177.504,18.907,152.548
C04997=1095.157,253.715,-76.318,177.500,18.905,152.548
C04998=1095.150,253.466,-76.290,177.497,18.903,152.548
C04999=1095.145,253.217,-76.263,177.494,18.902,152.548
C05000=1095.139,252.969,-76.236,177.491,18.900,152.549
C05001=1095.134,252.720,-76.209,177.487,18.898,152.549
C05002=1095.128,252.473,-76.182,177.485,18.896,152.549
C05003=1095.123,252.224,-76.155,177.481,18.894,152.549
C05004=1095.117,251.975,-76.127,177.478,18.892,152.549
C05005=1095.112,251.726,-76.100,177.475,18.891,152.549
C05006=1095.106,251.478,-76.074,177.472,18.889,152.550
C05007=1095.101,251.230,-76.046,177.469,18.887,152.550
C05008=1095.095,250.982,-76.019,177.466,18.886,152.550
C05009=1095.090,250.733,-75.992,177.462,18.884,152.550
C05010=1095.084,250.485,-75.965,177.459,18.882,152.550
C05011=1095.078,250.236,-75.938,177.456,18.880,152.550
C05012=1095.071,249.873,-75.898,177.451,18.877,152.551
C05013=1095.063,249.509,-75.859,177.447,18.875,152.551
C05014=1095.054,249.145,-75.820,177.443,18.873,152.551
C05015=1095.045,248.782,-75.780,177.438,18.869,152.551
C05016=1095.040,248.533,-75.753,177.435,18.868,152.552
C05017=1095.035,248.285,-75.726,177.432,18.866,152.552
C05018=1095.030,248.036,-75.699,177.428,18.864,152.552
C05019=1095.024,247.788,-75.672,177.425,18.863,152.552
C05020=1095.018,247.539,-75.646,177.422,18.861,152.552
C05021=1095.013,247.291,-75.618,177.418,18.859,152.553
C05022=1095.007,247.042,-75.592,177.416,18.857,152.553
C05023=1095.002,246.793,-75.566,177.412,18.856,152.553
C05024=1094.996,246.545,-75.539,177.409,18.854,152.553
C05025=1094.991,246.296,-75.512,177.406,18.852,152.553
C05026=1094.985,246.048,-75.485,177.403,18.851,152.554
C05027=1094.979,245.800,-75.459,177.399,18.849,152.554
C05028=1094.974,245.551,-75.432,177.397,18.847,152.554
C05029=1094.969,245.303,-75.405,177.393,18.845,152.554
C05030=1094.963,245.054,-75.378,177.391,18.844,152.554
C05031=1094.957,244.805,-75.352,177.387,18.842,152.554
C05032=1094.952,244.557,-75.325,177.384,18.840,152.555
C05033=1094.946,244.309,-75.299,177.381,18.839,152.555
C05034=1094.940,244.060,-75.272,177.378,18.837,152.555
C05035=1094.935,243.812,-75.245,177.374,18.835,152.555
C05036=1094.929,243.563,-75.219,177.372,18.833,152.555
C05037=1094.924,243.314,-75.192,177.368,18.832,152.556
C05038=1094.918,243.066,-75.166,177.365,18.830,152.556
C05039=1094.912,242.818,-75.139,177.362,18.828,152.556
C05040=1094.907,242.569,-75.113,177.358,18.826,152.556
C05041=1094.901,242.320,-75.086,177.356,18.825,152.556
C05042=1094.895,242.072,-75.060,177.352,18.823,152.557
C05043=1094.890,241.823,-75.034,177.349,18.821,152.557
C05044=1094.884,241.574,-75.007,177.346,18.820,152.557
C05045=1094.878,241.326,-74.981,177.343,18.818,152.557
C05046=1094.873,241.077,-74.955,177.340,18.817,152.557
C05047=1094.867,240.829,-74.928,177.337,18.815,152.558
C05048=1094.861,240.580,-74.901,177.333,18.813,152.558
C05049=1094.856,240.331,-74.875,177.330,18.812,152.558
C05050=1094.850,240.083,-74.849,177.327,18.810,152.558
C05051=1094.844,239.834,-74.823,177.324,18.809,152.559
C05052=1094.839,239.586,-74.796,177.321,18.807,152.559
C05053=1094.833,239.337,-74.770,177.317,18.805,152.559
C05054=1094.827,239.088,-74.744,177.315,18.803,152.559
C05055=1094.822,238.840,-74.717,177.311,18.802,152.559
C05056=1094.816,238.591,-74.691,177.308,18.801,152.560
C05057=1094.811,238.343,-74.665,177.305,18.798,152.560
C05058=1094.806,238.094,-74.639,177.302,18.797,152.560
C05059=1094.799,237.846,-74.613,177.299,18.795,152.560
C05060=1094.794,237.597,-74.587,177.295,18.794,152.560
C05061=1094.788,237.348,-74.561,177.293,18.792,152.561
C05062=1094.782,237.100,-74.534,177.289,18.790,152.561
C05063=1094.777,236.851,-74.508,177.287,18.789,152.561
C05064=1094.768,236.481,-74.469,177.281,18.786,152.561
C05065=1094.761,236.111,-74.431,177.277,18.784,152.562
C05066=1094.752,235.740,-74.392,177.273,18.782,152.562
C05067=1094.744,235.370,-74.353,177.267,18.779,152.562
C05068=1094.738,235.121,-74.327,177.265,18.778,152.562
C05069=1094.732,234.873,-74.301,177.261,18.776,152.563
C05070=1094.727,234.624,-74.275,177.259,18.774,152.563
C05071=1094.722,234.376,-74.249,177.255,18.772,152.563
C05072=1094.716,234.127,-74.223,177.252,18.771,152.563
C05073=1094.710,233.879,-74.197,177.249,18.769,152.564
C05074=1094.704,233.630,-74.171,177.245,18.767,152.564
C05075=1094.699,233.381,-74.145,177.243,18.766,152.564
C05076=1094.694,233.132,-74.120,177.239,18.764,152.564
C05077=1094.687,232.884,-74.094,177.236,18.763,152.564
C05078=1094.682,232.635,-74.068,177.233,18.761,152.565
C05079=1094.676,232.386,-74.042,177.230,18.760,152.565
C05080=1094.671,232.137,-74.016,177.227,18.758,152.565
C05081=1094.665,231.889,-73.991,177.224,18.757,152.565
C05082=1094.660,231.641,-73.964,177.221,18.755,152.565
C05083=1094.654,231.392,-73.938,177.217,18.753,152.566
C05084=1094.648,231.143,-73.913,177.215,18.752,152.566
C05085=1094.643,230.895,-73.887,177.211,18.750,152.566
C05086=1094.638,230.646,-73.861,177.208,18.749,152.566
C05087=1094.631,230.397,-73.836,177.205,18.747,152.566
C05088=1094.626,230.148,-73.810,177.202,18.745,152.567
C05089=1094.621,229.900,-73.785,177.199,18.744,152.567
C05090=1094.615,229.651,-73.759,177.196,18.742,152.567
C05091=1094.609,229.402,-73.733,177.192,18.741,152.567
C05092=1094.603,229.154,-73.708,177.190,18.739,152.568
C05093=1094.598,228.906,-73.682,177.186,18.737,152.568
C05094=1094.592,228.657,-73.657,177.184,18.736,152.568
C05095=1094.587,228.408,-73.631,177.180,18.734,152.568
C05096=1094.580,228.159,-73.606,177.177,18.733,152.569
C05097=1094.576,227.911,-73.580,177.174,18.731,152.569
C05098=1094.569,227.662,-73.555,177.171,18.730,152.569
C05099=1094.564,227.413,-73.529,177.168,18.728,152.569
C05100=1094.558,227.165,-73.504,177.165,18.727,152.569
C05101=1094.553,226.916,-73.478,177.162,18.725,152.570
C05102=1094.547,226.668,-73.453,177.159,18.724,152.570
C05103=1094.542,226.419,-73.427,177.155,18.722,152.570
C05104=1094.536,226.171,-73.402,177.153,18.721,152.570
C05105=1094.530,225.922,-73.376,177.149,18.719,152.570
C05106=1094.525,225.673,-73.352,177.147,18.718,152.571
C05107=1094.519,225.424,-73.326,177.143,18.716,152.571
C05108=1094.513,225.175,-73.300,177.140,18.715,152.571
C05109=1094.508,224.927,-73.275,177.137,18.713,152.571
C05110=1094.502,224.679,-73.250,177.134,18.711,152.572
C05111=1094.496,224.429,-73.225,177.131,18.710,152.572
C05112=1094.491,224.181,-73.199,177.128,18.708,152.572
C05113=1094.485,223.932,-73.174,177.124,18.707,152.572
C05114=1094.480,223.684,-73.148,177.122,18.705,152.573
C05115=1094.474,223.435,-73.124,177.118,18.703,152.573
C05116=1094.465,223.056,-73.085,177.114,18.701,152.573
C05117=1094.457,222.677,-73.046,177.109,18.699,152.573
C05118=1094.449,222.298,-73.008,177.104,18.696,152.574
C05119=1094.440,221.919,-72.969,177.100,18.694,152.574
C05120=1094.435,221.670,-72.945,177.096,18.692,152.574
C05121=1094.429,221.422,-72.919,177.093,18.691,152.575
C05122=1094.424,221.173,-72.895,177.090,18.689,152.575
C05123=1094.418,220.924,-72.870,177.087,18.688,152.575
C05124=1094.411,220.676,-72.844,177.084,18.686,152.575
C05125=1094.407,220.427,-72.819,177.081,18.685,152.576
C05126=1094.401,220.178,-72.794,177.078,18.684,152.576
C05127=1094.395,219.929,-72.770,177.075,18.682,152.576
C05128=1094.389,219.681,-72.744,177.072,18.681,152.576
C05129=1094.384,219.432,-72.720,177.069,18.679,152.576
C05130=1094.378,219.183,-72.694,177.066,18.678,152.577
C05131=1094.372,218.935,-72.669,177.062,18.676,152.577
C05132=1094.367,218.686,-72.645,177.060,18.675,152.577
C05133=1094.361,218.437,-72.619,177.056,18.673,152.577
C05134=1094.355,218.189,-72.595,177.053,18.672,152.578
C05135=1094.350,217.939,-72.570,177.050,18.670,152.578
C05136=1094.345,217.691,-72.545,177.047,18.668,152.578
C05137=1094.339,217.442,-72.520,177.044,18.667,152.578
C05138=1094.333,217.194,-72.495,177.041,18.666,152.579
C05139=1094.327,216.945,-72.471,177.038,18.664,152.579
C05140=1094.322,216.697,-72.446,177.035,18.663,152.579
C05141=1094.316,216.447,-72.421,177.032,18.661,152.579
C05142=1094.311,216.198,-72.396,177.029,18.659,152.579
C05143=1094.306,215.950,-72.371,177.026,18.658,152.580
C05144=1094.300,215.701,-72.347,177.022,18.656,152.580
C05145=1094.294,215.453,-72.322,177.020,18.655,152.580
C05146=1094.288,215.204,-72.297,177.016,18.653,152.580
C05147=1094.283,214.955,-72.273,177.013,18.652,152.581
C05148=1094.277,214.706,-72.248,177.011,18.651,152.581
C05149=1094.271,214.458,-72.223,177.007,18.649,152.581
C05150=1094.267,214.209,-72.198,177.005,18.648,152.581
C05151=1094.261,213.960,-72.174,177.001,18.646,152.582
C05152=1094.256,213.711,-72.149,176.998,18.645,152.582
C05153=1094.249,213.463,-72.124,176.995,18.643,152.582
C05154=1094.244,213.214,-72.100,176.992,18.642,152.582
C05155=1094.238,212.965,-72.075,176.990,18.640,152.582
C05156=1094.233,212.716,-72.051,176.986,18.638,152.583
C05157=1094.227,212.468,-72.026,176.983,18.637,152.583
C05158=1094.221,212.219,-72.001,176.980,18.635,152.583
C05159=1094.216,211.970,-71.977,176.977,18.634,152.583
C05160=1094.211,211.722,-71.953,176.973,18.633,152.584
C05161=1094.205,211.472,-71.928,176.971,18.631,152.584
C05162=1094.200,211.224,-71.904,176.968,18.630,152.584
C05163=1094.193,210.975,-71.880,176.965,18.628,152.584
C05164=1094.187,210.727,-71.855,176.962,18.627,152.585
C05165=1094.182,210.478,-71.831,176.958,18.625,152.585
C05166=1094.176,210.229,-71.806,176.956,18.624,152.585
C05167=1094.171,209.980,-71.782,176.953,18.623,152.585
C05168=1094.162,209.605,-71.745,176.948,18.620,152.586
C05169=1094.154,209.230,-71.708,176.943,18.618,152.586
C05170=1094.145,208.854,-71.672,176.939,18.616,152.586
C05171=1094.137,208.480,-71.635,176.934,18.613,152.587
C05172=1094.114,207.464,-71.538,176.878,18.589,152.592
C05173=1094.108,207.214,-71.513,176.875,18.588,152.592
C05174=1094.103,206.966,-71.489,176.872,18.588,152.593
C05175=1094.097,206.717,-71.466,176.869,18.587,152.593
C05176=1094.092,206.468,-71.441,176.866,18.587,152.594
C05177=1094.086,206.220,-71.417,176.863,18.586,152.594
C05178=1094.080,205.970,-71.394,176.860,18.585,152.594
C05179=1094.075,205.721,-71.370,176.856,18.585,152.595
C05180=1094.070,205.473,-71.345,176.853,18.584,152.595
C05181=1094.064,205.225,-71.322,176.849,18.584,152.596
C05182=1094.059,204.975,-71.298,176.846,18.583,152.596
C05183=1094.052,204.727,-71.275,176.843,18.582,152.597
C05184=1094.047,204.478,-71.250,176.840,18.582,152.597
C05185=1094.042,204.229,-71.226,176.837,18.581,152.598
C05186=1094.036,203.980,-71.203,176.834,18.581,152.598
C05187=1094.031,203.731,-71.179,176.831,18.580,152.598
C05188=1094.025,203.483,-71.156,176.828,18.580,152.599
C05189=1094.019,203.234,-71.131,176.824,18.578,152.599
C05190=1094.014,202.985,-71.108,176.821,18.578,152.600
C05191=1094.008,202.736,-71.084,176.818,18.577,152.600
C05192=1094.002,202.487,-71.061,176.815,18.577,152.601
C05193=1093.997,202.239,-71.036,176.812,18.577,152.601
C05194=1093.991,201.990,-71.014,176.809,18.576,152.602
C05195=1093.986,201.741,-70.989,176.805,18.576,152.602
C05196=1093.979,201.491,-70.966,176.802,18.575,152.603
C05197=1093.973,201.243,-70.942,176.799,18.575,152.603
C05198=1093.968,200.994,-70.919,176.796,18.574,152.603
C05199=1093.962,200.746,-70.895,176.793,18.573,152.604
C05200=1093.957,200.497,-70.872,176.790,18.573,152.604
C05201=1093.951,200.248,-70.848,176.786,18.572,152.605
C05202=1093.945,199.999,-70.825,176.783,18.572,152.605
C05203=1093.939,199.750,-70.800,176.780,18.571,152.606
C05204=1093.934,199.501,-70.777,176.777,18.570,152.606
C05205=1093.928,199.252,-70.754,176.774,18.570,152.607
C05206=1093.923,199.004,-70.730,176.771,18.569,152.607
C05207=1093.917,198.755,-70.707,176.767,18.569,152.608
C05208=1093.911,198.507,-70.684,176.764,18.568,152.608
C05209=1093.906,198.257,-70.660,176.761,18.568,152.608
C05210=1093.900,198.008,-70.637,176.758,18.567,152.609
C05211=1093.894,197.760,-70.613,176.755,18.567,152.609
C05212=1093.889,197.511,-70.590,176.752,18.566,152.610
C05213=1093.883,197.262,-70.567,176.749,18.566,152.610
C05214=1093.877,197.014,-70.543,176.746,18.565,152.611
C05215=1093.872,196.764,-70.519,176.743,18.564,152.611
C05216=1093.866,196.515,-70.496,176.740,18.564,152.612
C05217=1093.860,196.266,-70.473,176.737,18.563,152.612
C05218=1093.854,196.018,-70.450,176.734,18.563,152.612
C05219=1093.849,195.769,-70.426,176.730,18.561,152.613
C05220=1093.844,195.520,-70.403,176.727,18.561,152.613
C05221=1093.838,195.271,-70.380,176.724,18.560,152.614
C05222=1093.833,195.022,-70.356,176.721,18.560,152.614
C05223=1093.827,194.773,-70.333,176.718,18.559,152.615
C05224=1093.821,194.524,-70.310,176.715,18.559,152.615
C05225=1093.815,194.275,-70.287,176.712,18.558,152.616
C05226=1093.810,194.026,-70.264,176.709,18.557,152.616
C05227=1093.804,193.778,-70.240,176.706,18.557,152.616
C05228=1093.799,193.529,-70.217,176.702,18.557,152.617
C05229=1093.793,193.280,-70.194,176.699,18.556,152.617
C05230=1093.787,193.031,-70.171,176.696,18.555,152.618
C05231=1093.782,192.782,-70.148,176.693,18.554,152.618
C05232=1093.777,192.534,-70.125,176.690,18.554,152.619
C05233=1093.770,192.258,-70.099,176.687,18.554,152.619
C05234=1093.764,191.983,-70.074,176.683,18.552,152.619
C05235=1093.758,191.707,-70.048,176.680,18.552,152.620
C05236=1093.752,191.432,-70.023,176.677,18.551,152.620
C05237=1093.747,191.183,-69.999,176.674,18.551,152.621
C05238=1093.741,190.934,-69.976,176.671,18.550,152.621
C05239=1093.735,190.685,-69.953,176.668,18.550,152.622
C05240=1093.729,190.436,-69.930,176.664,18.549,152.622
C05241=1093.724,190.188,-69.908,176.661,18.548,152.623
C05242=1093.719,189.939,-69.884,176.658,18.547,152.623
C05243=1093.713,189.690,-69.861,176.655,18.546,152.623
C05244=1093.708,189.441,-69.839,176.652,18.546,152.624
C05245=1093.702,189.192,-69.816,176.649,18.545,152.624
C05246=1093.697,188.943,-69.793,176.646,18.544,152.625
C05247=1093.691,188.694,-69.770,176.643,18.544,152.625
C05248=1093.685,188.445,-69.747,176.640,18.543,152.626
C05249=1093.681,188.196,-69.724,176.637,18.543,152.626
C05250=1093.675,187.948,-69.701,176.634,18.542,152.626
C05251=1093.669,187.699,-69.678,176.631,18.541,152.627
C05252=1093.664,187.450,-69.655,176.628,18.541,152.627
C05253=1093.658,187.201,-69.632,176.625,18.540,152.628
C05254=1093.653,186.952,-69.610,176.622,18.539,152.628
C05255=1093.647,186.703,-69.587,176.619,18.539,152.628
C05256=1093.642,186.454,-69.564,176.616,18.538,152.629
C05257=1093.637,186.205,-69.541,176.613,18.537,152.629
C05258=1093.631,185.956,-69.518,176.610,18.537,152.630
C05259=1093.626,185.707,-69.496,176.607,18.536,152.630
C05260=1093.620,185.458,-69.473,176.604,18.535,152.630
C05261=1093.615,185.210,-69.450,176.601,18.534,152.631
C05262=1093.609,184.961,-69.427,176.598,18.534,152.631
C05263=1093.603,184.712,-69.404,176.595,18.534,152.632
C05264=1093.597,184.463,-69.383,176.592,18.533,152.632
C05265=1093.591,184.214,-69.360,176.589,18.532,152.633
C05266=1093.586,183.965,-69.337,176.586,18.531,152.633
C05267=1093.580,183.717,-69.314,176.583,18.531,152.633
C05268=1093.574,183.467,-69.292,176.580,18.531,152.634
C05269=1093.568,183.218,-69.270,176.577,18.530,152.634
C05270=1093.563,182.970,-69.247,176.574,18.530,152.635
C05271=1093.557,182.720,-69.224,176.571,18.529,152.635
C05272=1093.551,182.471,-69.202,176.568,18.528,152.635
C05273=1093.546,182.223,-69.179,176.565,18.528,152.636
C05274=1093.540,181.974,-69.157,176.562,18.527,152.636
C05275=1093.535,181.725,-69.134,176.559,18.527,152.637
C05276=1093.528,181.476,-69.112,176.556,18.526,152.637
C05277=1093.523,181.227,-69.090,176.553,18.525,152.638
C05278=1093.517,180.978,-69.067,176.550,18.525,152.638
C05279=1093.512,180.729,-69.045,176.547,18.524,152.638
C05280=1093.506,180.480,-69.023,176.544,18.523,152.639
C05281=1093.500,180.231,-69.000,176.541,18.523,152.639
C05282=1093.494,179.982,-68.977,176.538,18.522,152.640
C05283=1093.488,179.733,-68.955,176.535,18.522,152.640
C05284=1093.483,179.485,-68.933,176.532,18.521,152.641
C05285=1093.477,179.236,-68.910,176.529,18.520,152.641
C05286=1093.471,178.987,-68.889,176.526,18.520,152.641
C05287=1093.466,178.738,-68.866,176.523,18.519,152.642
C05288=1093.461,178.489,-68.844,176.520,18.518,152.642
C05289=1093.454,178.240,-68.821,176.517,18.518,152.643
C05290=1093.449,177.991,-68.799,176.514,18.517,152.643
C05291=1093.443,177.741,-68.777,176.512,18.517,152.643
C05292=1093.438,177.493,-68.755,176.509,18.516,152.644
C05293=1093.432,177.244,-68.733,176.506,18.515,152.644
C05294=1093.426,176.995,-68.710,176.503,18.515,152.645
C05295=1093.421,176.746,-68.689,176.500,18.514,152.645
C05296=1093.415,176.498,-68.666,176.497,18.513,152.645
C05297=1093.409,176.222,-68.641,176.494,18.513,152.646
C05298=1093.403,175.946,-68.617,176.490,18.511,152.646
C05299=1093.396,175.670,-68.592,176.487,18.511,152.647
C05300=1093.390,175.394,-68.568,176.484,18.511,152.647
C05301=1093.384,175.145,-68.545,176.481,18.510,152.648
C05302=1093.379,174.896,-68.523,176.478,18.509,152.648
C05303=1093.373,174.647,-68.502,176.475,18.509,152.648
C05304=1093.368,174.398,-68.479,176.472,18.507,152.649
C05305=1093.362,174.149,-68.457,176.469,18.507,152.649
C05306=1093.357,173.900,-68.435,176.466,18.506,152.649
C05307=1093.351,173.651,-68.413,176.463,18.505,152.650
C05308=1093.345,173.402,-68.391,176.460,18.505,152.650
C05309=1093.340,173.153,-68.369,176.457,18.504,152.651
C05310=1093.334,172.904,-68.347,176.455,18.504,152.651
C05311=1093.329,172.655,-68.325,176.452,18.503,152.651
C05312=1093.323,172.407,-68.303,176.449,18.502,152.652
C05313=1093.317,172.157,-68.281,176.446,18.502,152.652
C05314=1093.312,171.908,-68.259,176.443,18.501,152.653
C05315=1093.306,171.659,-68.237,176.440,18.500,152.653
C05316=1093.301,171.410,-68.215,176.437,18.499,152.653
C05317=1093.295,171.162,-68.193,176.434,18.499,152.654
C05318=1093.289,170.912,-68.171,176.431,18.498,152.654
C05319=1093.284,170.664,-68.149,176.428,18.497,152.655
C05320=1093.278,170.414,-68.127,176.425,18.496,152.655
C05321=1093.273,170.166,-68.106,176.422,18.495,152.655
C05322=1093.267,169.916,-68.084,176.420,18.495,152.656
C05323=1093.262,169.668,-68.062,176.417,18.495,152.656
C05324=1093.257,169.418,-68.040,176.414,18.494,152.656
C05325=1093.251,169.170,-68.019,176.411,18.493,152.657
C05326=1093.245,168.921,-67.996,176.409,18.492,152.657
C05327=1093.240,168.672,-67.975,176.406,18.491,152.657
C05328=1093.234,168.423,-67.953,176.403,18.491,152.658
C05329=1093.229,168.174,-67.931,176.400,18.490,152.658
C05330=1093.223,167.925,-67.909,176.397,18.489,152.659
C05331=1093.218,167.676,-67.888,176.394,18.488,152.659
C05332=1093.212,167.427,-67.866,176.392,18.488,152.659
C05333=1093.207,167.178,-67.844,176.389,18.487,152.660
C05334=1093.201,166.929,-67.822,176.386,18.486,152.660
C05335=1093.196,166.680,-67.801,176.383,18.486,152.660
C05336=1093.190,166.431,-67.779,176.380,18.484,152.661
C05337=1093.185,166.182,-67.757,176.377,18.484,152.661
C05338=1093.179,165.932,-67.736,176.374,18.483,152.661
C05339=1093.174,165.684,-67.714,176.371,18.482,152.662
C05340=1093.168,165.434,-67.693,176.368,18.481,152.662
C05341=1093.163,165.186,-67.671,176.366,18.481,152.663
C05342=1093.157,164.937,-67.650,176.364,18.480,152.663
C05343=1093.152,164.688,-67.627,176.361,18.479,152.663
C05344=1093.147,164.439,-67.606,176.358,18.479,152.664
C05345=1093.140,164.190,-67.585,176.355,18.477,152.664
C05346=1093.136,163.941,-67.563,176.352,18.477,152.664
C05347=1093.130,163.691,-67.542,176.349,18.476,152.665
C05348=1093.125,163.442,-67.520,176.346,18.475,152.665
C05349=1093.119,163.194,-67.499,176.343,18.474,152.665
C05350=1093.113,162.945,-67.477,176.341,18.474,152.666
C05351=1093.108,162.696,-67.455,176.338,18.473,152.666
C05352=1093.103,162.447,-67.435,176.335,18.472,152.666
C05353=1093.098,162.197,-67.412,176.332,18.471,152.667
C05354=1093.092,161.949,-67.391,176.329,18.471,152.667
C05355=1093.086,161.700,-67.369,176.327,18.469,152.667
C05356=1093.081,161.451,-67.348,176.324,18.469,152.668
C05357=1093.076,161.202,-67.327,176.321,18.468,152.668
C05358=1093.070,160.952,-67.305,176.319,18.467,152.668
C05359=1093.064,160.704,-67.284,176.316,18.467,152.669
C05360=1093.058,160.454,-67.263,176.313,18.466,152.669
C05361=1093.052,160.178,-67.239,176.310,18.465,152.669
C05362=1093.046,159.901,-67.216,176.307,18.464,152.670
C05363=1093.039,159.626,-67.192,176.303,18.463,152.670
C05364=1093.034,159.349,-67.168,176.300,18.462,152.671
C05365=1093.028,159.101,-67.147,176.297,18.462,152.671
C05366=1093.022,158.852,-67.126,176.295,18.461,152.671
C05367=1093.017,158.602,-67.105,176.292,18.460,152.672
C05368=1093.011,158.354,-67.084,176.290,18.459,152.672
C05369=1093.005,158.105,-67.062,176.287,18.459,152.672
C05370=1093.000,157.855,-67.042,176.284,18.458,152.673
C05371=1092.995,157.607,-67.020,176.281,18.457,152.673
C05372=1092.989,157.357,-66.999,176.278,18.456,152.673
C05373=1092.983,157.108,-66.978,176.276,18.455,152.674
C05374=1092.978,156.860,-66.956,176.273,18.455,152.674
C05375=1092.972,156.610,-66.935,176.270,18.454,152.674
C05376=1092.966,156.361,-66.914,176.267,18.453,152.675
C05377=1092.961,156.112,-66.893,176.264,18.452,152.675
C05378=1092.955,155.863,-66.872,176.261,18.451,152.675
C05379=1092.950,155.614,-66.851,176.259,18.451,152.676
C05380=1092.944,155.365,-66.830,176.257,18.450,152.676
C05381=1092.938,155.116,-66.809,176.254,18.449,152.677
C05382=1092.933,154.867,-66.788,176.251,18.448,152.677
C05383=1092.927,154.618,-66.767,176.248,18.447,152.677
C05384=1092.921,154.369,-66.746,176.245,18.446,152.677
C05385=1092.916,154.120,-66.725,176.243,18.446,152.678
C05386=1092.910,153.871,-66.704,176.240,18.445,152.678
C05387=1092.905,153.621,-66.683,176.237,18.444,152.679
C05388=1092.899,153.372,-66.662,176.234,18.444,152.679
C05389=1092.894,153.124,-66.641,176.231,18.443,152.679
C05390=1092.889,152.875,-66.621,176.228,18.442,152.680
C05391=1092.882,152.625,-66.599,176.227,18.441,152.680
C05392=1092.877,152.376,-66.578,176.224,18.441,152.680
C05393=1092.872,152.127,-66.558,176.221,18.439,152.680
C05394=1092.865,151.878,-66.537,176.218,18.438,152.681
C05395=1092.860,151.629,-66.516,176.215,18.438,152.681
C05396=1092.854,151.380,-66.496,176.212,18.436,152.681
C05397=1092.849,151.131,-66.474,176.210,18.436,152.682
C05398=1092.843,150.882,-66.453,176.207,18.435,152.682
C05399=1092.838,150.633,-66.433,176.204,18.435,152.682
C05400=1092.832,150.384,-66.412,176.202,18.433,152.683
C05401=1092.827,150.135,-66.391,176.199,18.433,152.683
C05402=1092.821,149.885,-66.370,176.197,18.432,152.683
C05403=1092.815,149.637,-66.349,176.194,18.431,152.684
C05404=1092.810,149.388,-66.329,176.191,18.430,152.684
C05405=1092.804,149.139,-66.308,176.188,18.429,152.684
C05406=1092.799,148.890,-66.288,176.185,18.429,152.685
C05407=1092.793,148.640,-66.266,176.183,18.428,152.685
C05408=1092.788,148.391,-66.246,176.181,18.427,152.685
C05409=1092.782,148.142,-66.226,176.178,18.426,152.686
C05410=1092.776,147.893,-66.205,176.175,18.425,152.686
C05411=1092.771,147.643,-66.184,176.172,18.424,152.686
C05412=1092.765,147.395,-66.163,176.170,18.424,152.687
C05413=1092.759,147.146,-66.143,176.167,18.423,152.687
C05414=1092.754,146.897,-66.122,176.164,18.422,152.687
C05415=1092.748,146.648,-66.102,176.161,18.421,152.687
C05416=1092.742,146.398,-66.082,176.158,18.420,152.688
C05417=1092.737,146.149,-66.061,176.157,18.419,152.688
C05418=1092.731,145.900,-66.040,176.154,18.418,152.688
C05419=1092.726,145.652,-66.019,176.151,18.418,152.689
C05420=1092.720,145.403,-65.999,176.148,18.417,152.689
C05421=1092.714,145.153,-65.978,176.145,18.416,152.689
C05422=1092.709,144.904,-65.958,176.143,18.415,152.690
C05423=1092.703,144.655,-65.938,176.140,18.414,152.690
C05424=1092.697,144.406,-65.917,176.137,18.413,152.690
C05425=1092.691,144.130,-65.894,176.135,18.412,152.691
C05426=1092.685,143.853,-65.872,176.132,18.411,152.691
C05427=1092.679,143.577,-65.849,176.129,18.411,152.691
C05428=1092.673,143.300,-65.826,176.126,18.409,152.692
C05429=1092.667,143.052,-65.806,176.123,18.409,152.692
C05430=1092.662,142.802,-65.786,176.120,18.408,152.692
C05431=1092.656,142.553,-65.765,176.118,18.406,152.693
C05432=1092.650,142.304,-65.745,176.116,18.406,152.693
C05433=1092.644,142.055,-65.724,176.113,18.405,152.693
C05434=1092.639,141.806,-65.704,176.110,18.404,152.693
C05435=1092.633,141.556,-65.684,176.107,18.403,152.694
C05436=1092.628,141.307,-65.664,176.105,18.402,152.694
C05437=1092.622,141.058,-65.644,176.102,18.402,152.694
C05438=1092.617,140.809,-65.623,176.100,18.400,152.695
C05439=1092.612,140.560,-65.603,176.097,18.399,152.695
C05440=1092.606,140.311,-65.583,176.094,18.398,152.695
C05441=1092.600,140.062,-65.562,176.092,18.398,152.696
C05442=1092.594,139.812,-65.542,176.089,18.397,152.696
C05443=1092.589,139.563,-65.521,176.087,18.396,152.696
C05444=1092.583,139.315,-65.501,176.084,18.395,152.696
C05445=1092.578,139.065,-65.482,176.082,18.394,152.697
C05446=1092.572,138.816,-65.462,176.079,18.393,152.697
C05447=1092.566,138.567,-65.441,176.076,18.392,152.697
C05448=1092.560,138.318,-65.421,176.073,18.391,152.698
C05449=1092.555,138.069,-65.401,176.071,18.391,152.698
C05450=1092.550,137.819,-65.381,176.069,18.389,152.698
C05451=1092.544,137.570,-65.361,176.066,18.389,152.698
C05452=1092.538,137.322,-65.341,176.063,18.388,152.699
C05453=1092.533,137.072,-65.320,176.061,18.387,152.699
C05454=1092.527,136.824,-65.300,176.058,18.386,152.699
